// enums
Datatypes.RegisterDatatype(_eTcVn2dCodeSearchStrategy);
Datatypes.RegisterDatatype(_eTcVnAdaptiveThresholdMethod);
Datatypes.RegisterDatatype(_eTcVnBarcodeSearchDirection);
Datatypes.RegisterDatatype(_eTcVnBarcodeType);
Datatypes.RegisterDatatype(_eTcVnBlobCombination);
Datatypes.RegisterDatatype(_eTcVnBoostClassifierType);
Datatypes.RegisterDatatype(_eTcVnBorderInterpolationMethod);
Datatypes.RegisterDatatype(_eTcVnCalibrationPattern);
Datatypes.RegisterDatatype(_eTcVnCalibrationPatternOrigin);
Datatypes.RegisterDatatype(_eTcVnCameraState);
Datatypes.RegisterDatatype(_eTcVnClusteringAlgorithm);
Datatypes.RegisterDatatype(_eTcVnCodeDetectionModel);
Datatypes.RegisterDatatype(_eTcVnCodeType);
Datatypes.RegisterDatatype(_eTcVnColorMap);
Datatypes.RegisterDatatype(_eTcVnColorMapSize);
Datatypes.RegisterDatatype(_eTcVnColorSpaceTransform);
Datatypes.RegisterDatatype(_eTcVnColorTrainingMethod);
Datatypes.RegisterDatatype(_eTcVnConnectedComponentsAlgorithm);
Datatypes.RegisterDatatype(_eTcVnContainerExportFormat);
Datatypes.RegisterDatatype(_eTcVnContourApproximationMethod);
Datatypes.RegisterDatatype(_eTcVnContourRetrievalMode);
Datatypes.RegisterDatatype(_eTcVnContoursMatchComparisonMethod);
Datatypes.RegisterDatatype(_eTcVnDiffusivityTypeKAZE);
Datatypes.RegisterDatatype(_eTcVnDistanceTransformationLabel);
Datatypes.RegisterDatatype(_eTcVnDistanceTransformationMask);
Datatypes.RegisterDatatype(_eTcVnDistanceType);
Datatypes.RegisterDatatype(_eTcVnDrawMatchesFlags);
Datatypes.RegisterDatatype(_eTcVnDrawShape);
Datatypes.RegisterDatatype(_eTcVnEdgeDetectionAlgorithm);
Datatypes.RegisterDatatype(_eTcVnEdgeDirection);
Datatypes.RegisterDatatype(_eTcVnElementType);
Datatypes.RegisterDatatype(_eTcVnEstimationAlgorithm);
Datatypes.RegisterDatatype(_eTcVnExtremePointDirection);
Datatypes.RegisterDatatype(_eTcVnFeatureDescriptorTypeAKAZE);
Datatypes.RegisterDatatype(_eTcVnFeatureScalingType);
Datatypes.RegisterDatatype(_eTcVnFeatureScoreTypeORB);
Datatypes.RegisterDatatype(_eTcVnFilterDirection);
Datatypes.RegisterDatatype(_eTcVnFindTemplateWalshOptions);
Datatypes.RegisterDatatype(_eTcVnFlipAxis);
Datatypes.RegisterDatatype(_eTcVnFontType);
Datatypes.RegisterDatatype(_eTcVnHoughMethod);
Datatypes.RegisterDatatype(_eTcVnInitializableFunction);
Datatypes.RegisterDatatype(_eTcVnInterpolationType);
Datatypes.RegisterDatatype(_eTcVnKeypointDetectionTypeAGAST);
Datatypes.RegisterDatatype(_eTcVnKeypointDetectionTypeFAST);
Datatypes.RegisterDatatype(_eTcVnKnn);
Datatypes.RegisterDatatype(_eTcVnLineType);
Datatypes.RegisterDatatype(_eTcVnMatchTemplateWalshOptions);
Datatypes.RegisterDatatype(_eTcVnMorphologicalOperator);
Datatypes.RegisterDatatype(_eTcVnNbc);
Datatypes.RegisterDatatype(_eTcVnNormalizationType);
Datatypes.RegisterDatatype(_eTcVnOcrModelType);
Datatypes.RegisterDatatype(_eTcVnOcrOptions);
Datatypes.RegisterDatatype(_eTcVnOrientationMethod);
Datatypes.RegisterDatatype(_eTcVnPaddingMode);
Datatypes.RegisterDatatype(_eTcVnPixelConnectivity);
Datatypes.RegisterDatatype(_eTcVnPixelEncoding);
Datatypes.RegisterDatatype(_eTcVnPixelPackMode);
Datatypes.RegisterDatatype(_eTcVnPrototypeClusterer);
Datatypes.RegisterDatatype(_eTcVnRectangleIntersection);
Datatypes.RegisterDatatype(_eTcVnRotationAngle);
Datatypes.RegisterDatatype(_eTcVnRTrees);
Datatypes.RegisterDatatype(_eTcVnSignedNormalization);
Datatypes.RegisterDatatype(_eTcVnSolvePnPMethod);
Datatypes.RegisterDatatype(_eTcVnSta);
Datatypes.RegisterDatatype(_eTcVnStructuringElementShape);
Datatypes.RegisterDatatype(_eTcVnSvm);
Datatypes.RegisterDatatype(_eTcVnSvmKernelType);
Datatypes.RegisterDatatype(_eTcVnSvmSgdClassifierMarginType);
Datatypes.RegisterDatatype(_eTcVnSvmSgdClassifierType);
Datatypes.RegisterDatatype(_eTcVnTemplateMatchMethod);
Datatypes.RegisterDatatype(_eTcVnThresholdType);
Datatypes.RegisterDatatype(_eTcVnTimestamp);
Datatypes.RegisterDatatype(_eTcVnVectorCompareMethod);
Datatypes.RegisterDatatype(_eTcVnWorldCoordinateSystem);
Datatypes.RegisterDatatype(_eTcWatchdogAccumulationType);
Datatypes.RegisterDatatype(_gEV_CAMERA_STATE);
Datatypes.RegisterDatatype(_eTcVnDataLayout);
Datatypes.RegisterDatatype(_eTcVnReduceType);
Datatypes.RegisterDatatype(_eTcVnCircularityCalculationMethod);
Datatypes.RegisterDatatype(_eTcVnDataMatrixOptions);
Datatypes.RegisterDatatype(_eTcVnLayerNameType);
    
Datatypes.RegisterDatatype(_eTcVnComparisonOperator);
Datatypes.RegisterDatatype(_eTcVnDetectBarcodesWalshOptions);
Datatypes.RegisterDatatype(_eTcVnDetectPatternPointsOptions);
Datatypes.RegisterDatatype(_eTcVnDotCodeOptions);
Datatypes.RegisterDatatype(_eTcVnEdgeSelection);
Datatypes.RegisterDatatype(_eTcVnFindRoisMethod);
Datatypes.RegisterDatatype(_eTcVnJpegSampling);
Datatypes.RegisterDatatype(_eTcVnMergeRegionsOptions);
Datatypes.RegisterDatatype(_eTcVnPolarizedImageInterpolation);
Datatypes.RegisterDatatype(_eTcVnSalientFeaturesMethod);
// structs
Datatypes.RegisterDatatype(_gVSP_IMAGE_INFO);
Datatypes.RegisterDatatype(_gVSP_LEADER_PAYLOAD_IMAGE);
Datatypes.RegisterDatatype(_gVSP_PIXEL_FORMAT);
Datatypes.RegisterDatatype(_tcVnCameraCalibrationOptions);
Datatypes.RegisterDatatype(_tcVnCircularArc);
Datatypes.RegisterDatatype(_tcVnCodeGrades1D);
Datatypes.RegisterDatatype(_tcVnCodeGradesDM);
Datatypes.RegisterDatatype(_tcVnCodeGradesQR);
Datatypes.RegisterDatatype(_tcVnDMatch);
Datatypes.RegisterDatatype(_tcVnImageInfo);
Datatypes.RegisterDatatype(_tcVnKeyPoint);
//Datatypes.RegisterDatatype(_tcVnMatrix);
Datatypes.RegisterDatatype(_tcVnMoments);
Datatypes.RegisterDatatype(_tcVnParamsAGAST);
Datatypes.RegisterDatatype(_tcVnParamsAKAZE);
Datatypes.RegisterDatatype(_tcVnParamsBlobDetection);
Datatypes.RegisterDatatype(_tcVnParamsBRISK);
Datatypes.RegisterDatatype(_tcVnParamsFAST);
Datatypes.RegisterDatatype(_tcVnParamsGFTT);
Datatypes.RegisterDatatype(_tcVnParamsKAZE);
Datatypes.RegisterDatatype(_tcVnParamsMSER);
Datatypes.RegisterDatatype(_tcVnParamsORB);
Datatypes.RegisterDatatype(_tcVnParamsSB);
Datatypes.RegisterDatatype(_tcVnPixelFormat);
Datatypes.RegisterDatatype(_tcVnRectangle_DINT);
Datatypes.RegisterDatatype(_tcVnRectangle_UDINT);
Datatypes.RegisterDatatype(_tcVnRotatedRectangle);
Datatypes.RegisterDatatype(_tcVnSize2_REAL);

Datatypes.RegisterDatatype(_gVCP_ADDRESS_VALUE_PAIR);
Datatypes.RegisterDatatype(_tcVnSize2_DINT);
Datatypes.RegisterDatatype(_tcVnParamsFindRois);
Datatypes.RegisterDatatype(_tcVnParamsWalshBarcodeDetection);
// interfaces
Datatypes.RegisterDatatype(_iTcVnImage);
Datatypes.RegisterDatatype(_iTcVnContainer);
Datatypes.RegisterDatatype(_iTcVnDisplayableImage);
END_METHOD

END_FUNCTION_BLOCK

// ---- Datatypes/Aliases/_GVCP_REGISTER_VALUE.TcPOU
{attribute 'linkalways'}
{attribute 'no_explicit_call' := 'This FB is a CLASS and must be accessed using methods or properties'}
{attribute 'enable_dynamic_creation'}
FUNCTION_BLOCK _GVCP_REGISTER_VALUE EXTENDS AliasDatatypeBase
VAR
	localData : GVCP_REGISTER_VALUE;
	activeData : REFERENCE TO GVCP_REGISTER_VALUE REF= localData;
	aliasBaseDatatype : _UDINT(0);
END_VAR

PROPERTY PUBLIC Address : PVOID
GET
Address := ADR(activeData);
END_GET
END_PROPERTY

METHOD PUBLIC ClearReference
VAR_INPUT
END_VAR
activeData REF= localData;
SetBaseDatatypeReference();
END_METHOD

METHOD PUBLIC Clone : I_Datatype
VAR
    pClone : POINTER TO _GVCP_REGISTER_VALUE;
END_VAR
pClone := __NEW(_GVCP_REGISTER_VALUE(InitialValue := Value));
IF pClone = 0 THEN
    RETURN;
END_IF
pClone^.TryCopyFrom(THIS^);
Clone := pClone^;
END_METHOD

METHOD FB_init : BOOL
VAR_INPUT
	bInitRetains : BOOL; // if TRUE, the retain variables are initialized (warm start / cold start)
	bInCopyCode : BOOL;  // if TRUE, the instance afterwards gets moved into the copy code (online change)
	InitialValue : GVCP_REGISTER_VALUE := 0;
END_VAR
localData := InitialValue;
SetBaseDatatypeReference();
AddBaseDatatype(aliasBaseDatatype);
END_METHOD

PROPERTY PUBLIC Identifier : T_MAXSTRING
GET
Identifier := 'GVCP_REGISTER_VALUE';
END_GET
END_PROPERTY

METHOD PUBLIC MakeReferenceTo
VAR_INPUT
	ReferenceTarget : REFERENCE TO GVCP_REGISTER_VALUE;
END_VAR
activeData REF= ReferenceTarget;
SetBaseDatatypeReference();
END_METHOD

METHOD PROTECTED SetBaseDatatypeReference
VAR_INPUT
END_VAR
aliasBaseDatatype.MakeReferenceTo(activeData);
END_METHOD

PROPERTY PUBLIC Size : UDINT
GET
Size := SIZEOF(activeData);
END_GET
END_PROPERTY

METHOD TryMakeReferenceTo : BOOL
VAR_INPUT
	Target : I_Datatype;
END_VAR
VAR
	pTargetData : POINTER TO GVCP_REGISTER_VALUE;
END_VAR
IF NOT IsEquivalentTo(Target) THEN
	RETURN;
END_IF

pTargetData := Target.Address;
activeData REF= pTargetData^;
SetBaseDatatypeReference();
TryMakeReferenceTo := TRUE;
END_METHOD

PROPERTY PUBLIC Value : REFERENCE TO GVCP_REGISTER_VALUE
GET
Value REF= activeData;
END_GET
END_PROPERTY

END_FUNCTION_BLOCK

// ---- Datatypes/Enums/_ETcVnComparisonOperator.TcPOU
{attribute 'linkalways'}
{attribute 'no_explicit_call' := 'This FB is a CLASS and must be accessed using methods or properties'}
{attribute 'enable_dynamic_creation'}
FUNCTION_BLOCK _ETcVnComparisonOperator EXTENDS EnumDatatypeBase
VAR
	localData : ETcVnComparisonOperator;
	activeData : REFERENCE TO ETcVnComparisonOperator;
	enumBaseDatatype : _INT(localData);
END_VAR

METHOD PRIVATE AddLocalEnumeration
VAR_INPUT
	Enumeration : T_MAXSTRING;
	Value : ETcVnComparisonOperator;
END_VAR
AddEnumeration(Enumeration, Value);
END_METHOD

PROPERTY PUBLIC Address : PVOID
GET
Address := ADR(activeData);
END_GET
END_PROPERTY

METHOD PUBLIC ClearReference
VAR_INPUT
END_VAR
activeData REF= localData;
SetBaseDatatypeReference();
END_METHOD

METHOD PUBLIC Clone : I_Datatype
VAR
    pClone : POINTER TO _ETcVnComparisonOperator;
END_VAR
pClone := __NEW(_ETcVnComparisonOperator(InitialValue := Value));
IF pClone = 0 THEN
    RETURN;
END_IF
Clone := pClone^;
END_METHOD

METHOD FB_init : BOOL
VAR_INPUT
	bInitRetains : BOOL; // if TRUE, the retain variables are initialized (warm start / cold start)
	bInCopyCode : BOOL;  // if TRUE, the instance afterwards gets moved into the copy code (online change)
	InitialValue : ETcVnComparisonOperator;
END_VAR
localData := InitialValue;
AddBaseDatatype(enumBaseDatatype);
ClearReference();

AddLocalEnumeration('TCVN_CO_LESS', ETcVnComparisonOperator.TCVN_CO_LESS);
AddLocalEnumeration('TCVN_CO_GREATER', ETcVnComparisonOperator.TCVN_CO_GREATER);
END_METHOD

PROPERTY PUBLIC Identifier : T_MAXSTRING
GET
Identifier := 'ETcVnComparisonOperator';
END_GET
END_PROPERTY

METHOD IsEnumeratorValueEqual : BOOL
VAR_INPUT
	Enumerator : I_KeyValueForwardEnumerator;
END_VAR
VAR
	storedValue : ETcVnComparisonOperator;
END_VAR
IF NOT Enumerator.TryGet(storedValue) THEN
	RETURN;
END_IF

IsEnumeratorValueEqual := storedValue = activeData;
END_METHOD

METHOD PUBLIC MakeReferenceTo
VAR_INPUT
	ReferenceTarget : REFERENCE TO ETcVnComparisonOperator;
END_VAR
activeData REF= ReferenceTarget;
SetBaseDatatypeReference();
END_METHOD

METHOD PROTECTED SetBaseDatatypeReference
VAR_INPUT
END_VAR
enumBaseDatatype.MakeReferenceTo(activeData);
END_METHOD

PROPERTY PUBLIC Size : UDINT
GET
Size := SIZEOF(activeData);
END_GET
END_PROPERTY

METHOD TryMakeReferenceTo : BOOL
VAR_INPUT
	Target : I_Datatype;
END_VAR
VAR
	pTargetData : POINTER TO ETcVnComparisonOperator;
END_VAR
IF NOT IsEquivalentTo(Target) THEN
	RETURN;
END_IF

pTargetData := Target.Address;
activeData REF= pTargetData^;
SetBaseDatatypeReference();
TryMakeReferenceTo := TRUE;
END_METHOD

PROPERTY PUBLIC Value : ETcVnComparisonOperator
GET
Value := activeData;
END_GET
SET
activeData := Value;
END_SET
END_PROPERTY

END_FUNCTION_BLOCK

// ---- Datatypes/Enums/_ETcVnDetectBarcodesWalshOptions.TcPOU
{attribute 'linkalways'}
{attribute 'no_explicit_call' := 'This FB is a CLASS and must be accessed using methods or properties'}
{attribute 'enable_dynamic_creation'}
FUNCTION_BLOCK _ETcVnDetectBarcodesWalshOptions EXTENDS EnumDatatypeBase
VAR
	localData : ETcVnDetectBarcodesWalshOptions;
	activeData : REFERENCE TO ETcVnDetectBarcodesWalshOptions;
	enumBaseDatatype : _UDINT(localData);
END_VAR

METHOD PRIVATE AddLocalEnumeration
VAR_INPUT
	Enumeration : T_MAXSTRING;
	Value : ETcVnDetectBarcodesWalshOptions;
END_VAR
AddEnumeration(Enumeration, Value);
END_METHOD

PROPERTY PUBLIC Address : PVOID
GET
Address := ADR(activeData);
END_GET
END_PROPERTY

METHOD PUBLIC ClearReference
VAR_INPUT
END_VAR
activeData REF= localData;
SetBaseDatatypeReference();
END_METHOD

METHOD PUBLIC Clone : I_Datatype
VAR
    pClone : POINTER TO _ETcVnDetectBarcodesWalshOptions;
END_VAR
pClone := __NEW(_ETcVnDetectBarcodesWalshOptions(InitialValue := Value));
IF pClone = 0 THEN
    RETURN;
END_IF
Clone := pClone^;
END_METHOD

METHOD FB_init : BOOL
VAR_INPUT
	bInitRetains : BOOL; // if TRUE, the retain variables are initialized (warm start / cold start)
	bInCopyCode : BOOL;  // if TRUE, the instance afterwards gets moved into the copy code (online change)
	InitialValue : ETcVnDetectBarcodesWalshOptions;
END_VAR
localData := InitialValue;
AddBaseDatatype(enumBaseDatatype);
ClearReference();

AddLocalEnumeration('TCVN_DBWO_HORIZONTAL', ETcVnDetectBarcodesWalshOptions.TCVN_DBWO_HORIZONTAL);
AddLocalEnumeration('TCVN_DBWO_VERTICAL', ETcVnDetectBarcodesWalshOptions.TCVN_DBWO_VERTICAL);
AddLocalEnumeration('TCVN_DBWO_DIAGONAL_45', ETcVnDetectBarcodesWalshOptions.TCVN_DBWO_DIAGONAL_45);
AddLocalEnumeration('TCVN_DBWO_DIAGONAL_135', ETcVnDetectBarcodesWalshOptions.TCVN_DBWO_DIAGONAL_135);
AddLocalEnumeration('TCVN_DBWO_ALL_DIRECTIONS', ETcVnDetectBarcodesWalshOptions.TCVN_DBWO_ALL_DIRECTIONS);
END_METHOD

PROPERTY PUBLIC Identifier : T_MAXSTRING
GET
Identifier := 'ETcVnDetectBarcodesWalshOptions';
END_GET
END_PROPERTY

METHOD IsEnumeratorValueEqual : BOOL
VAR_INPUT
	Enumerator : I_KeyValueForwardEnumerator;
END_VAR
VAR
	storedValue : ETcVnDetectBarcodesWalshOptions;
END_VAR
IF NOT Enumerator.TryGet(storedValue) THEN
	RETURN;
END_IF

IsEnumeratorValueEqual := storedValue = activeData;
END_METHOD

METHOD PUBLIC MakeReferenceTo
VAR_INPUT
	ReferenceTarget : REFERENCE TO ETcVnDetectBarcodesWalshOptions;
END_VAR
activeData REF= ReferenceTarget;
SetBaseDatatypeReference();
END_METHOD

METHOD PROTECTED SetBaseDatatypeReference
VAR_INPUT
END_VAR
enumBaseDatatype.MakeReferenceTo(activeData);
END_METHOD

PROPERTY PUBLIC Size : UDINT
GET
Size := SIZEOF(activeData);
END_GET
END_PROPERTY

METHOD TryMakeReferenceTo : BOOL
VAR_INPUT
	Target : I_Datatype;
END_VAR
VAR
	pTargetData : POINTER TO ETcVnDetectBarcodesWalshOptions;
END_VAR
IF NOT IsEquivalentTo(Target) THEN
	RETURN;
END_IF

pTargetData := Target.Address;
activeData REF= pTargetData^;
SetBaseDatatypeReference();
TryMakeReferenceTo := TRUE;
END_METHOD

PROPERTY PUBLIC Value : ETcVnDetectBarcodesWalshOptions
GET
Value := activeData;
END_GET
SET
activeData := Value;
END_SET
END_PROPERTY

END_FUNCTION_BLOCK

// ---- Datatypes/Enums/_ETcVnDetectPatternPointsOptions.TcPOU
{attribute 'linkalways'}
{attribute 'no_explicit_call' := 'This FB is a CLASS and must be accessed using methods or properties'}
{attribute 'enable_dynamic_creation'}
FUNCTION_BLOCK _ETcVnDetectPatternPointsOptions EXTENDS EnumDatatypeBase
VAR
	localData : ETcVnDetectPatternPointsOptions;
	activeData : REFERENCE TO ETcVnDetectPatternPointsOptions;
	enumBaseDatatype : _UDINT(localData);
END_VAR

METHOD PRIVATE AddLocalEnumeration
VAR_INPUT
	Enumeration : T_MAXSTRING;
	Value : ETcVnDetectPatternPointsOptions;
END_VAR
AddEnumeration(Enumeration, Value);
END_METHOD

PROPERTY PUBLIC Address : PVOID
GET
Address := ADR(activeData);
END_GET
END_PROPERTY

METHOD PUBLIC ClearReference
VAR_INPUT
END_VAR
activeData REF= localData;
SetBaseDatatypeReference();
END_METHOD

METHOD PUBLIC Clone : I_Datatype
VAR
    pClone : POINTER TO _ETcVnDetectPatternPointsOptions;
END_VAR
pClone := __NEW(_ETcVnDetectPatternPointsOptions(InitialValue := Value));
IF pClone = 0 THEN
    RETURN;
END_IF
Clone := pClone^;
END_METHOD

METHOD FB_init : BOOL
VAR_INPUT
	bInitRetains : BOOL; // if TRUE, the retain variables are initialized (warm start / cold start)
	bInCopyCode : BOOL;  // if TRUE, the instance afterwards gets moved into the copy code (online change)
	InitialValue : ETcVnDetectPatternPointsOptions;
END_VAR
localData := InitialValue;
AddBaseDatatype(enumBaseDatatype);
ClearReference();

AddLocalEnumeration('TCVN_DPPO_SYMMETRIC', ETcVnDetectPatternPointsOptions.TCVN_DPPO_SYMMETRIC);
AddLocalEnumeration('TCVN_DPPO_ASYMMETRIC', ETcVnDetectPatternPointsOptions.TCVN_DPPO_ASYMMETRIC);
AddLocalEnumeration('TCVN_DPPO_CLUSTERING', ETcVnDetectPatternPointsOptions.TCVN_DPPO_CLUSTERING);
END_METHOD

PROPERTY PUBLIC Identifier : T_MAXSTRING
GET
Identifier := 'ETcVnDetectPatternPointsOptions';
END_GET
END_PROPERTY

METHOD IsEnumeratorValueEqual : BOOL
VAR_INPUT
	Enumerator : I_KeyValueForwardEnumerator;
END_VAR
VAR
	storedValue : ETcVnDetectPatternPointsOptions;
END_VAR
IF NOT Enumerator.TryGet(storedValue) THEN
	RETURN;
END_IF

IsEnumeratorValueEqual := storedValue = activeData;
END_METHOD

METHOD PUBLIC MakeReferenceTo
VAR_INPUT
	ReferenceTarget : REFERENCE TO ETcVnDetectPatternPointsOptions;
END_VAR
activeData REF= ReferenceTarget;
SetBaseDatatypeReference();
END_METHOD

METHOD PROTECTED SetBaseDatatypeReference
VAR_INPUT
END_VAR
enumBaseDatatype.MakeReferenceTo(activeData);
END_METHOD

PROPERTY PUBLIC Size : UDINT
GET
Size := SIZEOF(activeData);
END_GET
END_PROPERTY

METHOD TryMakeReferenceTo : BOOL
VAR_INPUT
	Target : I_Datatype;
END_VAR
VAR
	pTargetData : POINTER TO ETcVnDetectPatternPointsOptions;
END_VAR
IF NOT IsEquivalentTo(Target) THEN
	RETURN;
END_IF

pTargetData := Target.Address;
activeData REF= pTargetData^;
SetBaseDatatypeReference();
TryMakeReferenceTo := TRUE;
END_METHOD

PROPERTY PUBLIC Value : ETcVnDetectPatternPointsOptions
GET
Value := activeData;
END_GET
SET
activeData := Value;
END_SET
END_PROPERTY

END_FUNCTION_BLOCK

// ---- Datatypes/Enums/_ETcVnDotCodeOptions.TcPOU
{attribute 'linkalways'}
{attribute 'no_explicit_call' := 'This FB is a CLASS and must be accessed using methods or properties'}
{attribute 'enable_dynamic_creation'}
FUNCTION_BLOCK _ETcVnDotCodeOptions EXTENDS EnumDatatypeBase
VAR
	localData : ETcVnDotCodeOptions;
	activeData : REFERENCE TO ETcVnDotCodeOptions;
	enumBaseDatatype : _ULINT(localData);
END_VAR

METHOD PRIVATE AddLocalEnumeration
VAR_INPUT
	Enumeration : T_MAXSTRING;
	Value : ETcVnDotCodeOptions;
END_VAR
AddEnumeration(Enumeration, Value);
END_METHOD

PROPERTY PUBLIC Address : PVOID
GET
Address := ADR(activeData);
END_GET
END_PROPERTY

METHOD PUBLIC ClearReference
VAR_INPUT
END_VAR
activeData REF= localData;
SetBaseDatatypeReference();
END_METHOD

METHOD PUBLIC Clone : I_Datatype
VAR
    pClone : POINTER TO _ETcVnDotCodeOptions;
END_VAR
pClone := __NEW(_ETcVnDotCodeOptions(InitialValue := Value));
IF pClone = 0 THEN
    RETURN;
END_IF
Clone := pClone^;
END_METHOD

METHOD FB_init : BOOL
VAR_INPUT
	bInitRetains : BOOL; // if TRUE, the retain variables are initialized (warm start / cold start)
	bInCopyCode : BOOL;  // if TRUE, the instance afterwards gets moved into the copy code (online change)
	InitialValue : ETcVnDotCodeOptions;
END_VAR
localData := InitialValue;
AddBaseDatatype(enumBaseDatatype);
ClearReference();

AddLocalEnumeration('TCVN_DCO_DEFAULT', ETcVnDotCodeOptions.TCVN_DCO_DEFAULT);
AddLocalEnumeration('TCVN_DCO_BINARY_INPUT', ETcVnDotCodeOptions.TCVN_DCO_BINARY_INPUT);
AddLocalEnumeration('TCVN_DCO_DETECTBLOBS', ETcVnDotCodeOptions.TCVN_DCO_DETECTBLOBS);
AddLocalEnumeration('TCVN_DCO_FILTERCONTOURS', ETcVnDotCodeOptions.TCVN_DCO_FILTERCONTOURS);
AddLocalEnumeration('TCVN_DCO_REGULAR_COLOR', ETcVnDotCodeOptions.TCVN_DCO_REGULAR_COLOR);
AddLocalEnumeration('TCVN_DCO_INVERTED_COLOR', ETcVnDotCodeOptions.TCVN_DCO_INVERTED_COLOR);
END_METHOD

PROPERTY PUBLIC Identifier : T_MAXSTRING
GET
Identifier := 'ETcVnDotCodeOptions';
END_GET
END_PROPERTY

METHOD IsEnumeratorValueEqual : BOOL
VAR_INPUT
	Enumerator : I_KeyValueForwardEnumerator;
END_VAR
VAR
	storedValue : ETcVnDotCodeOptions;
END_VAR
IF NOT Enumerator.TryGet(storedValue) THEN
	RETURN;
END_IF

IsEnumeratorValueEqual := storedValue = activeData;
END_METHOD

METHOD PUBLIC MakeReferenceTo
VAR_INPUT
	ReferenceTarget : REFERENCE TO ETcVnDotCodeOptions;
END_VAR
activeData REF= ReferenceTarget;
SetBaseDatatypeReference();
END_METHOD

METHOD PROTECTED SetBaseDatatypeReference
VAR_INPUT
END_VAR
enumBaseDatatype.MakeReferenceTo(activeData);
END_METHOD

PROPERTY PUBLIC Size : UDINT
GET
Size := SIZEOF(activeData);
END_GET
END_PROPERTY

METHOD TryMakeReferenceTo : BOOL
VAR_INPUT
	Target : I_Datatype;
END_VAR
VAR
	pTargetData : POINTER TO ETcVnDotCodeOptions;
END_VAR
IF NOT IsEquivalentTo(Target) THEN
	RETURN;
END_IF

pTargetData := Target.Address;
activeData REF= pTargetData^;
SetBaseDatatypeReference();
TryMakeReferenceTo := TRUE;
END_METHOD

PROPERTY PUBLIC Value : ETcVnDotCodeOptions
GET
Value := activeData;
END_GET
SET
activeData := Value;
END_SET
END_PROPERTY

END_FUNCTION_BLOCK

// ---- Datatypes/Enums/_ETcVnEdgeSelection.TcPOU
{attribute 'linkalways'}
{attribute 'no_explicit_call' := 'This FB is a CLASS and must be accessed using methods or properties'}
{attribute 'enable_dynamic_creation'}
FUNCTION_BLOCK _ETcVnEdgeSelection EXTENDS EnumDatatypeBase
VAR
	localData : ETcVnEdgeSelection;
	activeData : REFERENCE TO ETcVnEdgeSelection;
	enumBaseDatatype : _DINT(localData);
END_VAR

METHOD PRIVATE AddLocalEnumeration
VAR_INPUT
	Enumeration : T_MAXSTRING;
	Value : ETcVnEdgeSelection;
END_VAR
AddEnumeration(Enumeration, Value);
END_METHOD

PROPERTY PUBLIC Address : PVOID
GET
Address := ADR(activeData);
END_GET
END_PROPERTY

METHOD PUBLIC ClearReference
VAR_INPUT
END_VAR
activeData REF= localData;
SetBaseDatatypeReference();
END_METHOD

METHOD PUBLIC Clone : I_Datatype
VAR
    pClone : POINTER TO _ETcVnEdgeSelection;
END_VAR
pClone := __NEW(_ETcVnEdgeSelection(InitialValue := Value));
IF pClone = 0 THEN
    RETURN;
END_IF
Clone := pClone^;
END_METHOD

METHOD FB_init : BOOL
VAR_INPUT
	bInitRetains : BOOL; // if TRUE, the retain variables are initialized (warm start / cold start)
	bInCopyCode : BOOL;  // if TRUE, the instance afterwards gets moved into the copy code (online change)
	InitialValue : ETcVnEdgeSelection;
END_VAR
localData := InitialValue;
AddBaseDatatype(enumBaseDatatype);
ClearReference();

AddLocalEnumeration('TCVN_ES_RISING', ETcVnEdgeSelection.TCVN_ES_RISING);
AddLocalEnumeration('TCVN_ES_FALLING', ETcVnEdgeSelection.TCVN_ES_FALLING);
AddLocalEnumeration('TCVN_ES_ANY', ETcVnEdgeSelection.TCVN_ES_ANY);
END_METHOD

PROPERTY PUBLIC Identifier : T_MAXSTRING
GET
Identifier := 'ETcVnEdgeSelection';
END_GET
END_PROPERTY

METHOD IsEnumeratorValueEqual : BOOL
VAR_INPUT
	Enumerator : I_KeyValueForwardEnumerator;
END_VAR
VAR
	storedValue : ETcVnEdgeSelection;
END_VAR
IF NOT Enumerator.TryGet(storedValue) THEN
	RETURN;
END_IF

IsEnumeratorValueEqual := storedValue = activeData;
END_METHOD

METHOD PUBLIC MakeReferenceTo
VAR_INPUT
	ReferenceTarget : REFERENCE TO ETcVnEdgeSelection;
END_VAR
activeData REF= ReferenceTarget;
SetBaseDatatypeReference();
END_METHOD

METHOD PROTECTED SetBaseDatatypeReference
VAR_INPUT
END_VAR
enumBaseDatatype.MakeReferenceTo(activeData);
END_METHOD

PROPERTY PUBLIC Size : UDINT
GET
Size := SIZEOF(activeData);
END_GET
END_PROPERTY

METHOD TryMakeReferenceTo : BOOL
VAR_INPUT
	Target : I_Datatype;
END_VAR
VAR
	pTargetData : POINTER TO ETcVnEdgeSelection;
END_VAR
IF NOT IsEquivalentTo(Target) THEN
	RETURN;
END_IF

pTargetData := Target.Address;
activeData REF= pTargetData^;
SetBaseDatatypeReference();
TryMakeReferenceTo := TRUE;
END_METHOD

PROPERTY PUBLIC Value : ETcVnEdgeSelection
GET
Value := activeData;
END_GET
SET
activeData := Value;
END_SET
END_PROPERTY

END_FUNCTION_BLOCK

// ---- Datatypes/Enums/_ETcVnFindRoisMethod.TcPOU
{attribute 'linkalways'}
{attribute 'no_explicit_call' := 'This FB is a CLASS and must be accessed using methods or properties'}
{attribute 'enable_dynamic_creation'}
FUNCTION_BLOCK _ETcVnFindRoisMethod EXTENDS EnumDatatypeBase
VAR
	localData : ETcVnFindRoisMethod;
	activeData : REFERENCE TO ETcVnFindRoisMethod;
	enumBaseDatatype : _UDINT(localData);
END_VAR

METHOD PRIVATE AddLocalEnumeration
VAR_INPUT
	Enumeration : T_MAXSTRING;
	Value : ETcVnFindRoisMethod;
END_VAR
AddEnumeration(Enumeration, Value);
END_METHOD

PROPERTY PUBLIC Address : PVOID
GET
Address := ADR(activeData);
END_GET
END_PROPERTY

METHOD PUBLIC ClearReference
VAR_INPUT
END_VAR
activeData REF= localData;
SetBaseDatatypeReference();
END_METHOD

METHOD PUBLIC Clone : I_Datatype
VAR
    pClone : POINTER TO _ETcVnFindRoisMethod;
END_VAR
pClone := __NEW(_ETcVnFindRoisMethod(InitialValue := Value));
IF pClone = 0 THEN
    RETURN;
END_IF
Clone := pClone^;
END_METHOD

METHOD FB_init : BOOL
VAR_INPUT
	bInitRetains : BOOL; // if TRUE, the retain variables are initialized (warm start / cold start)
	bInCopyCode : BOOL;  // if TRUE, the instance afterwards gets moved into the copy code (online change)
	InitialValue : ETcVnFindRoisMethod;
END_VAR
localData := InitialValue;
AddBaseDatatype(enumBaseDatatype);
ClearReference();

AddLocalEnumeration('TCVN_FRM_GRID', ETcVnFindRoisMethod.TCVN_FRM_GRID);
AddLocalEnumeration('TCVN_FRM_CONNECTEDCOMPONENTS', ETcVnFindRoisMethod.TCVN_FRM_CONNECTEDCOMPONENTS);
END_METHOD

PROPERTY PUBLIC Identifier : T_MAXSTRING
GET
Identifier := 'ETcVnFindRoisMethod';
END_GET
END_PROPERTY

METHOD IsEnumeratorValueEqual : BOOL
VAR_INPUT
	Enumerator : I_KeyValueForwardEnumerator;
END_VAR
VAR
	storedValue : ETcVnFindRoisMethod;
END_VAR
IF NOT Enumerator.TryGet(storedValue) THEN
	RETURN;
END_IF

IsEnumeratorValueEqual := storedValue = activeData;
END_METHOD

METHOD PUBLIC MakeReferenceTo
VAR_INPUT
	ReferenceTarget : REFERENCE TO ETcVnFindRoisMethod;
END_VAR
activeData REF= ReferenceTarget;
SetBaseDatatypeReference();
END_METHOD

METHOD PROTECTED SetBaseDatatypeReference
VAR_INPUT
END_VAR
enumBaseDatatype.MakeReferenceTo(activeData);
END_METHOD

PROPERTY PUBLIC Size : UDINT
GET
Size := SIZEOF(activeData);
END_GET
END_PROPERTY

METHOD TryMakeReferenceTo : BOOL
VAR_INPUT
	Target : I_Datatype;
END_VAR
VAR
	pTargetData : POINTER TO ETcVnFindRoisMethod;
END_VAR
IF NOT IsEquivalentTo(Target) THEN
	RETURN;
END_IF

pTargetData := Target.Address;
activeData REF= pTargetData^;
SetBaseDatatypeReference();
TryMakeReferenceTo := TRUE;
END_METHOD

PROPERTY PUBLIC Value : ETcVnFindRoisMethod
GET
Value := activeData;
END_GET
SET
activeData := Value;
END_SET
END_PROPERTY

END_FUNCTION_BLOCK

// ---- Datatypes/Enums/_ETcVnJpegSampling.TcPOU
{attribute 'linkalways'}
{attribute 'no_explicit_call' := 'This FB is a CLASS and must be accessed using methods or properties'}
{attribute 'enable_dynamic_creation'}
FUNCTION_BLOCK _ETcVnJpegSampling EXTENDS EnumDatatypeBase
VAR
	localData : ETcVnJpegSampling;
	activeData : REFERENCE TO ETcVnJpegSampling;
	enumBaseDatatype : _DINT(localData);
END_VAR

METHOD PRIVATE AddLocalEnumeration
VAR_INPUT
	Enumeration : T_MAXSTRING;
	Value : ETcVnJpegSampling;
END_VAR
AddEnumeration(Enumeration, Value);
END_METHOD

PROPERTY PUBLIC Address : PVOID
GET
Address := ADR(activeData);
END_GET
END_PROPERTY

METHOD PUBLIC ClearReference
VAR_INPUT
END_VAR
activeData REF= localData;
SetBaseDatatypeReference();
END_METHOD

METHOD PUBLIC Clone : I_Datatype
VAR
    pClone : POINTER TO _ETcVnJpegSampling;
END_VAR
pClone := __NEW(_ETcVnJpegSampling(InitialValue := Value));
IF pClone = 0 THEN
    RETURN;
END_IF
Clone := pClone^;
END_METHOD

METHOD FB_init : BOOL
VAR_INPUT
	bInitRetains : BOOL; // if TRUE, the retain variables are initialized (warm start / cold start)
	bInCopyCode : BOOL;  // if TRUE, the instance afterwards gets moved into the copy code (online change)
	InitialValue : ETcVnJpegSampling;
END_VAR
localData := InitialValue;
AddBaseDatatype(enumBaseDatatype);
ClearReference();

AddLocalEnumeration('TCVN_JS_444', ETcVnJpegSampling.TCVN_JS_444);
AddLocalEnumeration('TCVN_JS_440', ETcVnJpegSampling.TCVN_JS_440);
AddLocalEnumeration('TCVN_JS_422', ETcVnJpegSampling.TCVN_JS_422);
AddLocalEnumeration('TCVN_JS_420', ETcVnJpegSampling.TCVN_JS_420);
AddLocalEnumeration('TCVN_JS_411', ETcVnJpegSampling.TCVN_JS_411);
AddLocalEnumeration('TCVN_JS_410', ETcVnJpegSampling.TCVN_JS_410);
END_METHOD

PROPERTY PUBLIC Identifier : T_MAXSTRING
GET
Identifier := 'ETcVnJpegSampling';
END_GET
END_PROPERTY

METHOD IsEnumeratorValueEqual : BOOL
VAR_INPUT
	Enumerator : I_KeyValueForwardEnumerator;
END_VAR
VAR
	storedValue : ETcVnJpegSampling;
END_VAR
IF NOT Enumerator.TryGet(storedValue) THEN
	RETURN;
END_IF

IsEnumeratorValueEqual := storedValue = activeData;
END_METHOD

METHOD PUBLIC MakeReferenceTo
VAR_INPUT
	ReferenceTarget : REFERENCE TO ETcVnJpegSampling;
END_VAR
activeData REF= ReferenceTarget;
SetBaseDatatypeReference();
END_METHOD

METHOD PROTECTED SetBaseDatatypeReference
VAR_INPUT
END_VAR
enumBaseDatatype.MakeReferenceTo(activeData);
END_METHOD

PROPERTY PUBLIC Size : UDINT
GET
Size := SIZEOF(activeData);
END_GET
END_PROPERTY

METHOD TryMakeReferenceTo : BOOL
VAR_INPUT
	Target : I_Datatype;
END_VAR
VAR
	pTargetData : POINTER TO ETcVnJpegSampling;
END_VAR
IF NOT IsEquivalentTo(Target) THEN
	RETURN;
END_IF

pTargetData := Target.Address;
activeData REF= pTargetData^;
SetBaseDatatypeReference();
TryMakeReferenceTo := TRUE;
END_METHOD

PROPERTY PUBLIC Value : ETcVnJpegSampling
GET
Value := activeData;
END_GET
SET
activeData := Value;
END_SET
END_PROPERTY

END_FUNCTION_BLOCK

// ---- Datatypes/Enums/_ETcVnMergeRegionsOptions.TcPOU
{attribute 'linkalways'}
{attribute 'no_explicit_call' := 'This FB is a CLASS and must be accessed using methods or properties'}
{attribute 'enable_dynamic_creation'}
FUNCTION_BLOCK _ETcVnMergeRegionsOptions EXTENDS EnumDatatypeBase
VAR
	localData : ETcVnMergeRegionsOptions;
	activeData : REFERENCE TO ETcVnMergeRegionsOptions;
	enumBaseDatatype : _ULINT(localData);
END_VAR

METHOD PRIVATE AddLocalEnumeration
VAR_INPUT
	Enumeration : T_MAXSTRING;
	Value : ETcVnMergeRegionsOptions;
END_VAR
AddEnumeration(Enumeration, Value);
END_METHOD

PROPERTY PUBLIC Address : PVOID
GET
Address := ADR(activeData);
END_GET
END_PROPERTY

METHOD PUBLIC ClearReference
VAR_INPUT
END_VAR
activeData REF= localData;
SetBaseDatatypeReference();
END_METHOD

METHOD PUBLIC Clone : I_Datatype
VAR
    pClone : POINTER TO _ETcVnMergeRegionsOptions;
END_VAR
pClone := __NEW(_ETcVnMergeRegionsOptions(InitialValue := Value));
IF pClone = 0 THEN
    RETURN;
END_IF
Clone := pClone^;
END_METHOD

METHOD FB_init : BOOL
VAR_INPUT
	bInitRetains : BOOL; // if TRUE, the retain variables are initialized (warm start / cold start)
	bInCopyCode : BOOL;  // if TRUE, the instance afterwards gets moved into the copy code (online change)
	InitialValue : ETcVnMergeRegionsOptions;
END_VAR
localData := InitialValue;
AddBaseDatatype(enumBaseDatatype);
ClearReference();

AddLocalEnumeration('TCVN_MRO_UPRIGHT_BOUNDING_RECT', ETcVnMergeRegionsOptions.TCVN_MRO_UPRIGHT_BOUNDING_RECT);
END_METHOD

PROPERTY PUBLIC Identifier : T_MAXSTRING
GET
Identifier := 'ETcVnMergeRegionsOptions';
END_GET
END_PROPERTY

METHOD IsEnumeratorValueEqual : BOOL
VAR_INPUT
	Enumerator : I_KeyValueForwardEnumerator;
END_VAR
VAR
	storedValue : ETcVnMergeRegionsOptions;
END_VAR
IF NOT Enumerator.TryGet(storedValue) THEN
	RETURN;
END_IF

IsEnumeratorValueEqual := storedValue = activeData;
END_METHOD

METHOD PUBLIC MakeReferenceTo
VAR_INPUT
	ReferenceTarget : REFERENCE TO ETcVnMergeRegionsOptions;
END_VAR
activeData REF= ReferenceTarget;
SetBaseDatatypeReference();
END_METHOD

METHOD PROTECTED SetBaseDatatypeReference
VAR_INPUT
END_VAR
enumBaseDatatype.MakeReferenceTo(activeData);
END_METHOD

PROPERTY PUBLIC Size : UDINT
GET
Size := SIZEOF(activeData);
END_GET
END_PROPERTY

METHOD TryMakeReferenceTo : BOOL
VAR_INPUT
	Target : I_Datatype;
END_VAR
VAR
	pTargetData : POINTER TO ETcVnMergeRegionsOptions;
END_VAR
IF NOT IsEquivalentTo(Target) THEN
	RETURN;
END_IF

pTargetData := Target.Address;
activeData REF= pTargetData^;
SetBaseDatatypeReference();
TryMakeReferenceTo := TRUE;
END_METHOD

PROPERTY PUBLIC Value : ETcVnMergeRegionsOptions
GET
Value := activeData;
END_GET
SET
activeData := Value;
END_SET
END_PROPERTY

END_FUNCTION_BLOCK

// ---- Datatypes/Enums/_ETcVnPolarizedImageInterpolation.TcPOU
{attribute 'linkalways'}
{attribute 'no_explicit_call' := 'This FB is a CLASS and must be accessed using methods or properties'}
{attribute 'enable_dynamic_creation'}
FUNCTION_BLOCK _ETcVnPolarizedImageInterpolation EXTENDS EnumDatatypeBase
VAR
	localData : ETcVnPolarizedImageInterpolation;
	activeData : REFERENCE TO ETcVnPolarizedImageInterpolation;
	enumBaseDatatype : _DINT(localData);
END_VAR

METHOD PRIVATE AddLocalEnumeration
VAR_INPUT
	Enumeration : T_MAXSTRING;
	Value : ETcVnPolarizedImageInterpolation;
END_VAR
AddEnumeration(Enumeration, Value);
END_METHOD

PROPERTY PUBLIC Address : PVOID
GET
Address := ADR(activeData);
END_GET
END_PROPERTY

METHOD PUBLIC ClearReference
VAR_INPUT
END_VAR
activeData REF= localData;
SetBaseDatatypeReference();
END_METHOD

METHOD PUBLIC Clone : I_Datatype
VAR
    pClone : POINTER TO _ETcVnPolarizedImageInterpolation;
END_VAR
pClone := __NEW(_ETcVnPolarizedImageInterpolation(InitialValue := Value));
IF pClone = 0 THEN
    RETURN;
END_IF
Clone := pClone^;
END_METHOD

METHOD FB_init : BOOL
VAR_INPUT
	bInitRetains : BOOL; // if TRUE, the retain variables are initialized (warm start / cold start)
	bInCopyCode : BOOL;  // if TRUE, the instance afterwards gets moved into the copy code (online change)
	InitialValue : ETcVnPolarizedImageInterpolation;
END_VAR
localData := InitialValue;
AddBaseDatatype(enumBaseDatatype);
ClearReference();

AddLocalEnumeration('TCVN_PII_NONE', ETcVnPolarizedImageInterpolation.TCVN_PII_NONE);
AddLocalEnumeration('TCVN_PII_NEAREST_NEIGHBOR', ETcVnPolarizedImageInterpolation.TCVN_PII_NEAREST_NEIGHBOR);
AddLocalEnumeration('TCVN_PII_BILINEAR', ETcVnPolarizedImageInterpolation.TCVN_PII_BILINEAR);
AddLocalEnumeration('TCVN_PII_BICUBIC', ETcVnPolarizedImageInterpolation.TCVN_PII_BICUBIC);
AddLocalEnumeration('TCVN_PII_LANCZOS4', ETcVnPolarizedImageInterpolation.TCVN_PII_LANCZOS4);
END_METHOD

PROPERTY PUBLIC Identifier : T_MAXSTRING
GET
Identifier := 'ETcVnPolarizedImageInterpolation';
END_GET
END_PROPERTY

METHOD IsEnumeratorValueEqual : BOOL
VAR_INPUT
	Enumerator : I_KeyValueForwardEnumerator;
END_VAR
VAR
	storedValue : ETcVnPolarizedImageInterpolation;
END_VAR
IF NOT Enumerator.TryGet(storedValue) THEN
	RETURN;
END_IF

IsEnumeratorValueEqual := storedValue = activeData;
END_METHOD

METHOD PUBLIC MakeReferenceTo
VAR_INPUT
	ReferenceTarget : REFERENCE TO ETcVnPolarizedImageInterpolation;
END_VAR
activeData REF= ReferenceTarget;
SetBaseDatatypeReference();
END_METHOD

METHOD PROTECTED SetBaseDatatypeReference
VAR_INPUT
END_VAR
enumBaseDatatype.MakeReferenceTo(activeData);
END_METHOD

PROPERTY PUBLIC Size : UDINT
GET
Size := SIZEOF(activeData);
END_GET
END_PROPERTY

METHOD TryMakeReferenceTo : BOOL
VAR_INPUT
	Target : I_Datatype;
END_VAR
VAR
	pTargetData : POINTER TO ETcVnPolarizedImageInterpolation;
END_VAR
IF NOT IsEquivalentTo(Target) THEN
	RETURN;
END_IF

pTargetData := Target.Address;
activeData REF= pTargetData^;
SetBaseDatatypeReference();
TryMakeReferenceTo := TRUE;
END_METHOD

PROPERTY PUBLIC Value : ETcVnPolarizedImageInterpolation
GET
Value := activeData;
END_GET
SET
activeData := Value;
END_SET
END_PROPERTY

END_FUNCTION_BLOCK

// ---- Datatypes/Enums/_ETcVnSalientFeaturesMethod.TcPOU
{attribute 'linkalways'}
{attribute 'no_explicit_call' := 'This FB is a CLASS and must be accessed using methods or properties'}
{attribute 'enable_dynamic_creation'}
FUNCTION_BLOCK _ETcVnSalientFeaturesMethod EXTENDS EnumDatatypeBase
VAR
	localData : ETcVnSalientFeaturesMethod;
	activeData : REFERENCE TO ETcVnSalientFeaturesMethod;
	enumBaseDatatype : _UDINT(localData);
END_VAR

METHOD PRIVATE AddLocalEnumeration
VAR_INPUT
	Enumeration : T_MAXSTRING;
	Value : ETcVnSalientFeaturesMethod;
END_VAR
AddEnumeration(Enumeration, Value);
END_METHOD

PROPERTY PUBLIC Address : PVOID
GET
Address := ADR(activeData);
END_GET
END_PROPERTY

METHOD PUBLIC ClearReference
VAR_INPUT
END_VAR
activeData REF= localData;
SetBaseDatatypeReference();
END_METHOD

METHOD PUBLIC Clone : I_Datatype
VAR
    pClone : POINTER TO _ETcVnSalientFeaturesMethod;
END_VAR
pClone := __NEW(_ETcVnSalientFeaturesMethod(InitialValue := Value));
IF pClone = 0 THEN
    RETURN;
END_IF
Clone := pClone^;
END_METHOD

METHOD FB_init : BOOL
VAR_INPUT
	bInitRetains : BOOL; // if TRUE, the retain variables are initialized (warm start / cold start)
	bInCopyCode : BOOL;  // if TRUE, the instance afterwards gets moved into the copy code (online change)
	InitialValue : ETcVnSalientFeaturesMethod;
END_VAR
localData := InitialValue;
AddBaseDatatype(enumBaseDatatype);
ClearReference();

AddLocalEnumeration('TCVN_SFM_WALSH_CODE', ETcVnSalientFeaturesMethod.TCVN_SFM_WALSH_CODE);
AddLocalEnumeration('TCVN_SFM_SOBEL', ETcVnSalientFeaturesMethod.TCVN_SFM_SOBEL);
END_METHOD

PROPERTY PUBLIC Identifier : T_MAXSTRING
GET
Identifier := 'ETcVnSalientFeaturesMethod';
END_GET
END_PROPERTY

METHOD IsEnumeratorValueEqual : BOOL
VAR_INPUT
	Enumerator : I_KeyValueForwardEnumerator;
END_VAR
VAR
	storedValue : ETcVnSalientFeaturesMethod;
END_VAR
IF NOT Enumerator.TryGet(storedValue) THEN
	RETURN;
END_IF

IsEnumeratorValueEqual := storedValue = activeData;
END_METHOD

METHOD PUBLIC MakeReferenceTo
VAR_INPUT
	ReferenceTarget : REFERENCE TO ETcVnSalientFeaturesMethod;
END_VAR
activeData REF= ReferenceTarget;
SetBaseDatatypeReference();
END_METHOD

METHOD PROTECTED SetBaseDatatypeReference
VAR_INPUT
END_VAR
enumBaseDatatype.MakeReferenceTo(activeData);
END_METHOD

PROPERTY PUBLIC Size : UDINT
GET
Size := SIZEOF(activeData);
END_GET
END_PROPERTY

METHOD TryMakeReferenceTo : BOOL
VAR_INPUT
	Target : I_Datatype;
END_VAR
VAR
	pTargetData : POINTER TO ETcVnSalientFeaturesMethod;
END_VAR
IF NOT IsEquivalentTo(Target) THEN
	RETURN;
END_IF

pTargetData := Target.Address;
activeData REF= pTargetData^;
SetBaseDatatypeReference();
TryMakeReferenceTo := TRUE;
END_METHOD

PROPERTY PUBLIC Value : ETcVnSalientFeaturesMethod
GET
Value := activeData;
END_GET
SET
activeData := Value;
END_SET
END_PROPERTY

END_FUNCTION_BLOCK

// ---- Datatypes/Structs/_GVCP_ADDRESS_VALUE_PAIR.TcPOU
{attribute 'linkalways'}
{attribute 'no_explicit_call' := 'This FB is a CLASS and must be accessed using methods or properties'}
{attribute 'enable_dynamic_creation'}
FUNCTION_BLOCK _GVCP_ADDRESS_VALUE_PAIR EXTENDS StructuredDatatypeBase
VAR
    localData : GVCP_ADDRESS_VALUE_PAIR;
    activeData : REFERENCE TO GVCP_ADDRESS_VALUE_PAIR REF= localData;
    _nAddress : _GVCP_REGISTER_ADDRESS(0);
    _nValue : _GVCP_REGISTER_VALUE(0);
END_VAR

PROPERTY PUBLIC Address : PVOID
GET
Address := ADR(activeData);
END_GET
END_PROPERTY

METHOD PUBLIC ClearReference
VAR_INPUT
END_VAR
activeData REF= localData;
SetMemberReference();
END_METHOD

METHOD PUBLIC Clone : I_Datatype
VAR
    pClone : POINTER TO _GVCP_ADDRESS_VALUE_PAIR;
END_VAR
pClone := __NEW(_GVCP_ADDRESS_VALUE_PAIR);
IF pClone = 0 THEN
    RETURN;
END_IF
pClone^.TryCopyFrom(THIS^);
Clone := pClone^;
END_METHOD

METHOD FB_init : BOOL
VAR_INPUT
	bInitRetains : BOOL; // if TRUE, the retain variables are initialized (warm start / cold start)
	bInCopyCode : BOOL;  // if TRUE, the instance afterwards gets moved into the copy code (online change)
END_VAR
SetMemberReference();
AddMember('nAddress', _nAddress);
AddMember('nValue', _nValue);
END_METHOD

PROPERTY PUBLIC Identifier : T_MAXSTRING
GET
Identifier := 'GVCP_ADDRESS_VALUE_PAIR';
END_GET
END_PROPERTY

METHOD PUBLIC MakeReferenceTo
VAR_INPUT
	ReferenceTarget : REFERENCE TO GVCP_ADDRESS_VALUE_PAIR;
END_VAR
activeData REF= ReferenceTarget;
SetMemberReference();
END_METHOD

PROPERTY PUBLIC nAddress : REFERENCE TO _GVCP_REGISTER_ADDRESS
GET
nAddress REF= _nAddress;
END_GET
END_PROPERTY

PROPERTY PUBLIC nValue : REFERENCE TO _GVCP_REGISTER_VALUE
GET
nValue REF= _nValue;
END_GET
END_PROPERTY

METHOD PROTECTED SetMemberReference
VAR_INPUT
END_VAR
_nAddress.MakeReferenceTo(activeData.nAddress);
_nValue.MakeReferenceTo(activeData.nValue);
END_METHOD

PROPERTY PUBLIC Size : UDINT
GET
Size := SIZEOF(activeData);
END_GET
END_PROPERTY

METHOD TryMakeReferenceTo : BOOL
VAR_INPUT
	Target : I_Datatype;
END_VAR
VAR
	pTargetData : POINTER TO GVCP_ADDRESS_VALUE_PAIR;
END_VAR
IF NOT IsEquivalentTo(Target) THEN
	RETURN;
END_IF

pTargetData := Target.Address;
activeData REF= pTargetData^;
SetMemberReference();
TryMakeReferenceTo := TRUE;
END_METHOD

PROPERTY PUBLIC Value : REFERENCE TO GVCP_ADDRESS_VALUE_PAIR
GET
Value REF= activeData;
END_GET
END_PROPERTY

END_FUNCTION_BLOCK

// ---- Datatypes/Structs/_TcVnSize2_DINT.TcPOU
{attribute 'linkalways'}
{attribute 'no_explicit_call' := 'This FB is a CLASS and must be accessed using methods or properties'}
{attribute 'enable_dynamic_creation'}
FUNCTION_BLOCK _TcVnSize2_DINT EXTENDS StructuredDatatypeBase
VAR
    localData : TcVnSize2_DINT;
    activeData : REFERENCE TO TcVnSize2_DINT REF= localData;
    _nWidth : _DINT(localData.nWidth);
    _nHeight : _DINT(localData.nHeight);
END_VAR

PROPERTY PUBLIC Address : PVOID
GET
Address := ADR(activeData);
END_GET
END_PROPERTY

METHOD PUBLIC ClearReference
VAR_INPUT
END_VAR
activeData REF= localData;
SetMemberReference();
END_METHOD

METHOD PUBLIC Clone : I_Datatype
VAR
    pClone : POINTER TO _TcVnSize2_DINT;
END_VAR
pClone := __NEW(_TcVnSize2_DINT);
IF pClone = 0 THEN
    RETURN;
END_IF
pClone^.TryCopyFrom(THIS^);
Clone := pClone^;
END_METHOD

METHOD FB_init : BOOL
VAR_INPUT
	bInitRetains : BOOL; // if TRUE, the retain variables are initialized (warm start / cold start)
	bInCopyCode : BOOL;  // if TRUE, the instance afterwards gets moved into the copy code (online change)
END_VAR
SetMemberReference();
AddMember('nWidth', _nWidth);
AddMember('nHeight', _nHeight);
END_METHOD

PROPERTY PUBLIC Identifier : T_MAXSTRING
GET
Identifier := 'TcVnSize2_DINT';
END_GET
END_PROPERTY

METHOD PUBLIC MakeReferenceTo
VAR_INPUT
	ReferenceTarget : REFERENCE TO TcVnSize2_DINT;
END_VAR
activeData REF= ReferenceTarget;
SetMemberReference();
END_METHOD

METHOD PROTECTED SetMemberReference
VAR_INPUT
END_VAR
_nWidth.MakeReferenceTo(activeData.nWidth);
_nHeight.MakeReferenceTo(activeData.nHeight);
END_METHOD

PROPERTY PUBLIC Size : UDINT
GET
Size := SIZEOF(activeData);
END_GET
END_PROPERTY

METHOD TryMakeReferenceTo : BOOL
VAR_INPUT
	Target : I_Datatype;
END_VAR
VAR
	pTargetData : POINTER TO TcVnSize2_DINT;
END_VAR
IF NOT IsEquivalentTo(Target) THEN
	RETURN;
END_IF

pTargetData := Target.Address;
activeData REF= pTargetData^;
SetMemberReference();
TryMakeReferenceTo := TRUE;
END_METHOD

PROPERTY PUBLIC Value : REFERENCE TO TcVnSize2_DINT
GET
Value REF= activeData;
END_GET
END_PROPERTY

PROPERTY PUBLIC nWidth : REFERENCE TO _DINT
GET
nWidth REF= _nWidth;
END_GET
END_PROPERTY

PROPERTY PUBLIC nHeight : REFERENCE TO _DINT
GET
nHeight REF= _nHeight;
END_GET
END_PROPERTY

END_FUNCTION_BLOCK

// ---- Datatypes/Structs/_TcVnParamsFindRois.TcPOU
{attribute 'linkalways'}
{attribute 'no_explicit_call' := 'This FB is a CLASS and must be accessed using methods or properties'}
{attribute 'enable_dynamic_creation'}
FUNCTION_BLOCK _TcVnParamsFindRois EXTENDS StructuredDatatypeBase
VAR
    localData : TcVnParamsFindRois := (stRoiSize := (nWidth := 416, nHeight := 416), fMinDensity := 0.2, fDetectionScaleFactor := 0.25, fMaxOversizeFraction := 1.0);
    activeData : REFERENCE TO TcVnParamsFindRois REF= localData;
    _stRoiSize : _TcVnSize2_DINT;
    _fMinDensity : _LREAL(localData.fMinDensity);
    _fDetectionScaleFactor : _LREAL(localData.fDetectionScaleFactor);
    _fMaxOversizeFraction : _LREAL(localData.fMaxOversizeFraction);
END_VAR

PROPERTY PUBLIC Address : PVOID
GET
Address := ADR(activeData);
END_GET
END_PROPERTY

METHOD PUBLIC ClearReference
VAR_INPUT
END_VAR
activeData REF= localData;
SetMemberReference();
END_METHOD

METHOD PUBLIC Clone : I_Datatype
VAR
    pClone : POINTER TO _TcVnParamsFindRois;
END_VAR
pClone := __NEW(_TcVnParamsFindRois);
IF pClone = 0 THEN
    RETURN;
END_IF
pClone^.TryCopyFrom(THIS^);
Clone := pClone^;
END_METHOD

METHOD FB_init : BOOL
VAR_INPUT
	bInitRetains : BOOL; // if TRUE, the retain variables are initialized (warm start / cold start)
	bInCopyCode : BOOL;  // if TRUE, the instance afterwards gets moved into the copy code (online change)
END_VAR
SetMemberReference();
AddMember('stRoiSize', _stRoiSize);
AddMember('fMinDensity', _fMinDensity);
AddMember('fDetectionScaleFactor', _fDetectionScaleFactor);
AddMember('fMaxOversizeFraction', _fMaxOversizeFraction);
END_METHOD

PROPERTY PUBLIC Identifier : T_MAXSTRING
GET
Identifier := 'TcVnParamsFindRois';
END_GET
END_PROPERTY

METHOD PUBLIC MakeReferenceTo
VAR_INPUT
	ReferenceTarget : REFERENCE TO TcVnParamsFindRois;
END_VAR
activeData REF= ReferenceTarget;
SetMemberReference();
END_METHOD

METHOD PROTECTED SetMemberReference
VAR_INPUT
END_VAR
_stRoiSize.MakeReferenceTo(activeData.stRoiSize);
_fMinDensity.MakeReferenceTo(activeData.fMinDensity);
_fDetectionScaleFactor.MakeReferenceTo(activeData.fDetectionScaleFactor);
_fMaxOversizeFraction.MakeReferenceTo(activeData.fMaxOversizeFraction);
END_METHOD

PROPERTY PUBLIC Size : UDINT
GET
Size := SIZEOF(activeData);
END_GET
END_PROPERTY

METHOD TryMakeReferenceTo : BOOL
VAR_INPUT
	Target : I_Datatype;
END_VAR
VAR
	pTargetData : POINTER TO TcVnParamsFindRois;
END_VAR
IF NOT IsEquivalentTo(Target) THEN
	RETURN;
END_IF

pTargetData := Target.Address;
activeData REF= pTargetData^;
SetMemberReference();
TryMakeReferenceTo := TRUE;
END_METHOD

PROPERTY PUBLIC Value : REFERENCE TO TcVnParamsFindRois
GET
Value REF= activeData;
END_GET
END_PROPERTY

PROPERTY PUBLIC stRoiSize : REFERENCE TO _TcVnSize2_DINT
GET
stRoiSize REF= _stRoiSize;
END_GET
END_PROPERTY

PROPERTY PUBLIC fMinDensity : REFERENCE TO _LREAL
GET
fMinDensity REF= _fMinDensity;
END_GET
END_PROPERTY

PROPERTY PUBLIC fDetectionScaleFactor : REFERENCE TO _LREAL
GET
fDetectionScaleFactor REF= _fDetectionScaleFactor;
END_GET
END_PROPERTY

PROPERTY PUBLIC fMaxOversizeFraction : REFERENCE TO _LREAL
GET
fMaxOversizeFraction REF= _fMaxOversizeFraction;
END_GET
END_PROPERTY

END_FUNCTION_BLOCK

// ---- Datatypes/Structs/_TcVnParamsWalshBarcodeDetection.TcPOU
{attribute 'linkalways'}
{attribute 'no_explicit_call' := 'This FB is a CLASS and must be accessed using methods or properties'}
{attribute 'enable_dynamic_creation'}
FUNCTION_BLOCK _TcVnParamsWalshBarcodeDetection EXTENDS StructuredDatatypeBase
VAR
    localData : TcVnParamsWalshBarcodeDetection := (nMaxBarDistance := 8, fMinAspectRatio := 1.0, fMaxAspectRatio := 5.0, nIntensityDifference := 100, nMinArea := -1, nChannelIndex := -1, nWalshFilterNum := 5, fOutlierReductionFactor := 1.0, fBarConnectionFactor := 1.0, fRegionFilterFactor := 1.0, fPostProcessingResizeFactor := 0.5, eInterpolationType := TCVN_IT_BILINEAR);
    activeData : REFERENCE TO TcVnParamsWalshBarcodeDetection REF= localData;
    _nMaxBarDistance : _UDINT(localData.nMaxBarDistance);
    _fMinAspectRatio : _REAL(localData.fMinAspectRatio);
    _fMaxAspectRatio : _REAL(localData.fMaxAspectRatio);
    _nIntensityDifference : _UDINT(localData.nIntensityDifference);
    _nMinArea : _DINT(localData.nMinArea);
    _nChannelIndex : _DINT(localData.nChannelIndex);
    _nWalshFilterNum : _UDINT(localData.nWalshFilterNum);
    _fOutlierReductionFactor : _REAL(localData.fOutlierReductionFactor);
    _fBarConnectionFactor : _REAL(localData.fBarConnectionFactor);
    _fRegionFilterFactor : _REAL(localData.fRegionFilterFactor);
    _fPostProcessingResizeFactor : _REAL(localData.fPostProcessingResizeFactor);
    _eInterpolationType : _ETcVnInterpolationType(localData.eInterpolationType);
END_VAR

PROPERTY PUBLIC Address : PVOID
GET
Address := ADR(activeData);
END_GET
END_PROPERTY

METHOD PUBLIC ClearReference
VAR_INPUT
END_VAR
activeData REF= localData;
SetMemberReference();
END_METHOD

METHOD PUBLIC Clone : I_Datatype
VAR
    pClone : POINTER TO _TcVnParamsWalshBarcodeDetection;
END_VAR
pClone := __NEW(_TcVnParamsWalshBarcodeDetection);
IF pClone = 0 THEN
    RETURN;
END_IF
pClone^.TryCopyFrom(THIS^);
Clone := pClone^;
END_METHOD

METHOD FB_init : BOOL
VAR_INPUT
	bInitRetains : BOOL; // if TRUE, the retain variables are initialized (warm start / cold start)
	bInCopyCode : BOOL;  // if TRUE, the instance afterwards gets moved into the copy code (online change)
END_VAR
SetMemberReference();
AddMember('nMaxBarDistance', _nMaxBarDistance);
AddMember('fMinAspectRatio', _fMinAspectRatio);
AddMember('fMaxAspectRatio', _fMaxAspectRatio);
AddMember('nIntensityDifference', _nIntensityDifference);
AddMember('nMinArea', _nMinArea);
AddMember('nChannelIndex', _nChannelIndex);
AddMember('nWalshFilterNum', _nWalshFilterNum);
AddMember('fOutlierReductionFactor', _fOutlierReductionFactor);
AddMember('fBarConnectionFactor', _fBarConnectionFactor);
AddMember('fRegionFilterFactor', _fRegionFilterFactor);
AddMember('fPostProcessingResizeFactor', _fPostProcessingResizeFactor);
AddMember('eInterpolationType', _eInterpolationType);
END_METHOD

PROPERTY PUBLIC Identifier : T_MAXSTRING
GET
Identifier := 'TcVnParamsWalshBarcodeDetection';
END_GET
END_PROPERTY

METHOD PUBLIC MakeReferenceTo
VAR_INPUT
	ReferenceTarget : REFERENCE TO TcVnParamsWalshBarcodeDetection;
END_VAR
activeData REF= ReferenceTarget;
SetMemberReference();
END_METHOD

METHOD PROTECTED SetMemberReference
VAR_INPUT
END_VAR
_nMaxBarDistance.MakeReferenceTo(activeData.nMaxBarDistance);
_fMinAspectRatio.MakeReferenceTo(activeData.fMinAspectRatio);
_fMaxAspectRatio.MakeReferenceTo(activeData.fMaxAspectRatio);
_nIntensityDifference.MakeReferenceTo(activeData.nIntensityDifference);
_nMinArea.MakeReferenceTo(activeData.nMinArea);
_nChannelIndex.MakeReferenceTo(activeData.nChannelIndex);
_nWalshFilterNum.MakeReferenceTo(activeData.nWalshFilterNum);
_fOutlierReductionFactor.MakeReferenceTo(activeData.fOutlierReductionFactor);
_fBarConnectionFactor.MakeReferenceTo(activeData.fBarConnectionFactor);
_fRegionFilterFactor.MakeReferenceTo(activeData.fRegionFilterFactor);
_fPostProcessingResizeFactor.MakeReferenceTo(activeData.fPostProcessingResizeFactor);
_eInterpolationType.MakeReferenceTo(activeData.eInterpolationType);
END_METHOD

PROPERTY PUBLIC Size : UDINT
GET
Size := SIZEOF(activeData);
END_GET
END_PROPERTY

METHOD TryMakeReferenceTo : BOOL
VAR_INPUT
	Target : I_Datatype;
END_VAR
VAR
	pTargetData : POINTER TO TcVnParamsWalshBarcodeDetection;
END_VAR
IF NOT IsEquivalentTo(Target) THEN
	RETURN;
END_IF

pTargetData := Target.Address;
activeData REF= pTargetData^;
SetMemberReference();
TryMakeReferenceTo := TRUE;
END_METHOD

PROPERTY PUBLIC Value : REFERENCE TO TcVnParamsWalshBarcodeDetection
GET
Value REF= activeData;
END_GET
END_PROPERTY

PROPERTY PUBLIC nMaxBarDistance : REFERENCE TO _UDINT
GET
nMaxBarDistance REF= _nMaxBarDistance;
END_GET
END_PROPERTY

PROPERTY PUBLIC fMinAspectRatio : REFERENCE TO _REAL
GET
fMinAspectRatio REF= _fMinAspectRatio;
END_GET
END_PROPERTY

PROPERTY PUBLIC fMaxAspectRatio : REFERENCE TO _REAL
GET
fMaxAspectRatio REF= _fMaxAspectRatio;
END_GET
END_PROPERTY

PROPERTY PUBLIC nIntensityDifference : REFERENCE TO _UDINT
GET
nIntensityDifference REF= _nIntensityDifference;
END_GET
END_PROPERTY

PROPERTY PUBLIC nMinArea : REFERENCE TO _DINT
GET
nMinArea REF= _nMinArea;
END_GET
END_PROPERTY

PROPERTY PUBLIC nChannelIndex : REFERENCE TO _DINT
GET
nChannelIndex REF= _nChannelIndex;
END_GET
END_PROPERTY

PROPERTY PUBLIC nWalshFilterNum : REFERENCE TO _UDINT
GET
nWalshFilterNum REF= _nWalshFilterNum;
END_GET
END_PROPERTY

PROPERTY PUBLIC fOutlierReductionFactor : REFERENCE TO _REAL
GET
fOutlierReductionFactor REF= _fOutlierReductionFactor;
END_GET
END_PROPERTY

PROPERTY PUBLIC fBarConnectionFactor : REFERENCE TO _REAL
GET
fBarConnectionFactor REF= _fBarConnectionFactor;
END_GET
END_PROPERTY

PROPERTY PUBLIC fRegionFilterFactor : REFERENCE TO _REAL
GET
fRegionFilterFactor REF= _fRegionFilterFactor;
END_GET
END_PROPERTY

PROPERTY PUBLIC fPostProcessingResizeFactor : REFERENCE TO _REAL
GET
fPostProcessingResizeFactor REF= _fPostProcessingResizeFactor;
END_GET
END_PROPERTY

PROPERTY PUBLIC eInterpolationType : REFERENCE TO _ETcVnInterpolationType
GET
eInterpolationType REF= _eInterpolationType;
END_GET
END_PROPERTY

END_FUNCTION_BLOCK

// ---- Extensions/PreExecutionCheck/PreExecutionCheckExtension.TcPOU
FUNCTION_BLOCK PreExecutionCheckExtension EXTENDS Extension
VAR
	parentAsPreCheckedNode : I_PreCheckedNode;
	preExecutionCheckFailedAlarm : PreExecutionCheckFailedAlarm(THIS^);
	enable : _BOOL(TRUE);
END_VAR

METHOD PUBLIC Check : BOOL
VAR_INPUT
END_VAR
VAR
	preExecutionChecks : PreExecutionChecks;
END_VAR
IF NOT enable.Value THEN
	IF preExecutionCheckFailedAlarm.Active THEN
		preExecutionCheckFailedAlarm.Clear();
	END_IF
	Check := TRUE;
	RETURN;
END_IF

parentAsPreCheckedNode.PreExecutionCheck(preExecutionChecks);
IF preExecutionChecks.Failed THEN
	preExecutionCheckFailedAlarm.Raise(preExecutionChecks.Reason);
	RETURN;
END_IF

preExecutionCheckFailedAlarm.Clear();
Check := TRUE;
END_METHOD

METHOD FB_init : BOOL
VAR_INPUT
	bInitRetains : BOOL; // if TRUE, the retain variables are initialized (warm start / cold start)
	bInCopyCode : BOOL;  // if TRUE, the instance afterwards gets moved into the copy code (online change)
	Name : T_MAXSTRING;
	Parent : I_HostExtensions;
END_VAR
AddParameter('enable', enable);

IF NOT __QUERYINTERFACE(Parent, parentAsPreCheckedNode) THEN
	RETURN;
END_IF
END_METHOD

END_FUNCTION_BLOCK

// ---- Extensions/WatchdogCheck/WatchdogCheckExtension.TcPOU
FUNCTION_BLOCK WatchdogCheckExtension EXTENDS Extension
VAR
	watchdogAlarm : FunctionFailedAlarm(THIS^);
	watchdogTimeInUs : _DINT(500000); // default
	hResult : HRESULT;
END_VAR

METHOD FB_init : BOOL
VAR_INPUT
	bInitRetains : BOOL; // if TRUE, the retain variables are initialized (warm start / cold start)
	bInCopyCode : BOOL;  // if TRUE, the instance afterwards gets moved into the copy code (online change)
	Name : T_MAXSTRING;
	Parent : I_HostExtensions;
END_VAR
AddParameter('watchdogTimeInUs', watchdogTimeInUs);
END_METHOD

METHOD PUBLIC Start
VAR_INPUT
END_VAR
watchdogAlarm.Clear();

IF watchdogTimeInUs.Value = 0 THEN
	RETURN;
END_IF

hResult := F_VN_StartRelWatchdog(watchdogTimeInUs.Value, S_OK);
END_METHOD

METHOD PUBLIC Stop
VAR_INPUT
END_VAR
hresult := F_VN_StopWatchdog(
	hrStartWatchdog := hresult);

IF FAILED(hresult) THEN
	watchdogAlarm.Raise('Watchdog', hresult);
END_IF
END_METHOD

END_FUNCTION_BLOCK

// ---- Functions/Checks/ContainersHaveMatchingNumberOfElements.TcPOU
FUNCTION ContainersHaveMatchingNumberOfElements : BOOL
VAR_INPUT
	Container1 : ITcVnContainer;
	Container2 : ITcVnContainer;
END_VAR
VAR
    elementNum1 : ULINT;
    elementNum2 : ULINT;
END_VAR

IF NOT IsValidContainer(Container1) THEN
	RETURN;
END_IF

IF NOT IsValidContainer(Container2) THEN
	RETURN;
END_IF

IF NOT SUCCEEDED(Container1.GetElementNum(elementNum1)) THEN
    RETURN;
END_IF

IF NOT SUCCEEDED(Container2.GetElementNum(elementNum2)) THEN
    RETURN;
END_IF

ContainersHaveMatchingNumberOfElements := (elementNum1 = elementNum2);

END_FUNCTION

// ---- Functions/Checks/IsValidContainer.TcPOU
FUNCTION IsValidContainer : BOOL
VAR_INPUT
    Container : ITcVnContainer;
END_VAR

IsValidContainer := Container <> 0;

END_FUNCTION

// ---- Functions/Checks/ImageHasCompatibleElementType.TcPOU
FUNCTION ImageHasCompatibleElementType : BOOL
VAR_INPUT
	Image : ITcVnImage;	
END_VAR
VAR_IN_OUT
	CompatibleElementTypes : ARRAY[*] OF ETcVnElementType;
END_VAR
VAR
	i : DINT;
END_VAR

IF NOT IsValidImage(Image) THEN
	RETURN;
END_IF

FOR i := LOWER_BOUND(CompatibleElementTypes, 1) TO UPPER_BOUND(CompatibleElementTypes, 1) DO
	IF ImageHasElementType(Image, CompatibleElementTypes[i]) THEN
		ImageHasCompatibleElementType := TRUE;
		RETURN;
	END_IF
END_FOR

END_FUNCTION

// ---- Functions/Checks/IsValidImage.TcPOU
FUNCTION IsValidImage : BOOL
VAR_INPUT
    Image : ITcVnImage;
END_VAR

IsValidImage := Image <> 0;

END_FUNCTION

// ---- Functions/Checks/ImageHasElementType.TcPOU
FUNCTION ImageHasElementType : BOOL
VAR_INPUT
	Image : ITcVnImage;
	ElementType : ETcVnElementType;
END_VAR

IF NOT IsValidImage(Image) THEN
	RETURN;
END_IF

ImageHasElementType := (ElementType = GetETcVnElementTypeFromImage(Image));

END_FUNCTION

// ---- Functions/Helpers/GetETcVnElementTypeFromImage.TcPOU
FUNCTION GetETcVnElementTypeFromImage : ETcVnElementType
VAR_INPUT
	sourceImage : ITcVnImage;
END_VAR
VAR
	pixelFormat : TcVnPixelFormat;
END_VAR

IF NOT IsValidImage(sourceImage) THEN
	RETURN;
END_IF

sourceImage.GetPixelFormat(pixelFormat);

IF pixelFormat.nElementSize = 8 AND NOT pixelFormat.bSigned THEN
	GetETcVnElementTypeFromImage := ETcVnElementType.TCVN_ET_USINT;
ELSIF pixelFormat.nElementSize = 8 AND pixelFormat.bSigned THEN
	GetETcVnElementTypeFromImage := ETcVnElementType.TCVN_ET_SINT;
ELSIF pixelFormat.nElementSize = 16 AND NOT pixelFormat.bSigned THEN
	GetETcVnElementTypeFromImage := ETcVnElementType.TCVN_ET_UINT;
ELSIF pixelFormat.nElementSize = 16 AND pixelFormat.bSigned THEN
	GetETcVnElementTypeFromImage := ETcVnElementType.TCVN_ET_INT;
ELSIF pixelFormat.nElementSize = 32 AND NOT pixelFormat.bFloat THEN
	GetETcVnElementTypeFromImage := ETcVnElementType.TCVN_ET_DINT;
ELSIF pixelFormat.nElementSize = 32 AND pixelFormat.bFloat THEN
	GetETcVnElementTypeFromImage := ETcVnElementType.TCVN_ET_REAL;
ELSIF pixelFormat.nElementSize = 64 THEN
	GetETcVnElementTypeFromImage := ETcVnElementType.TCVN_ET_LREAL;
ELSE
	GetETcVnElementTypeFromImage := ETcVnElementType.TCVN_ET_SAME_AS_SOURCE;
END_IF

END_FUNCTION

// ---- Functions/Checks/ImagesHaveMatchingChannels.TcPOU
FUNCTION ImagesHaveMatchingChannels : BOOL
VAR_INPUT
	Image1 : ITcVnImage;
	Image2 : ITcVnImage;
END_VAR
VAR
	pixelFormat1: TcVnPixelFormat;
	pixelFormat2: TcVnPixelFormat;
END_VAR

IF NOT IsValidImage(Image1) THEN
	RETURN;
END_IF

IF NOT IsValidImage(Image2) THEN
	RETURN;
END_IF

Image1.GetPixelFormat(pixelFormat1);
Image2.GetPixelFormat(pixelFormat2);

ImagesHaveMatchingChannels := (pixelFormat1.nChannels = pixelFormat2.nChannels);

END_FUNCTION

// ---- Functions/Checks/ContainersHaveMatchingTypes.TcPOU
FUNCTION ContainersHaveMatchingTypes : BOOL
VAR_INPUT
	Container1 : ITcVnContainer;
	Container2 : ITcVnContainer;
END_VAR
VAR
    guid1 : GUID;
    guid2 : GUID;
END_VAR

IF NOT IsValidContainer(Container1) THEN
	RETURN;
END_IF

IF NOT IsValidContainer(Container2) THEN
	RETURN;
END_IF

IF NOT SUCCEEDED(Container1.GetTypeGuid(guid1)) THEN
    RETURN;
END_IF

IF NOT SUCCEEDED(Container2.GetTypeGuid(guid2)) THEN
    RETURN;
END_IF

ContainersHaveMatchingTypes := GuidsEqualByVal(guid1, guid2);

END_FUNCTION

// ---- Functions/Checks/ImagesHaveMatchingPixelFormats.TcPOU
FUNCTION ImagesHaveMatchingPixelFormats : BOOL
VAR_INPUT
	Image1 : ITcVnImage;
	Image2 : ITcVnImage;
END_VAR
VAR
	pixelFormat_1: TcVnPixelFormat;
	pixelFormat_2: TcVnPixelFormat;
	pointer_1 : POINTER TO BYTE;
	pointer_2 : POINTER TO BYTE;
END_VAR

IF NOT IsValidImage(Image1) THEN
	RETURN;
END_IF

IF NOT IsValidImage(Image2) THEN
	RETURN;
END_IF

Image1.GetPixelFormat(pixelFormat_1);
Image2.GetPixelFormat(pixelFormat_2);

pointer_1 := ADR(pixelFormat_1);
pointer_2 := ADR(pixelFormat_2);

ImagesHaveMatchingPixelFormats := (MEMCMP(pointer_1, pointer_2, SIZEOF(pixelFormat_1)) = 0);

END_FUNCTION

// ---- Functions/Checks/IsImage1SizeEqualToImage2Size.TcPOU
FUNCTION IsImage1SizeEqualToImage2Size : BOOL
VAR_INPUT
    Image1 : ITcVnImage;
    Image2 : ITcVnImage;
END_VAR
VAR
    image1Width : UDINT;
    image1Height : UDINT;
    image2Width : UDINT;
    image2Height : UDINT;
END_VAR

IF NOT IsValidImage(Image1) THEN
    RETURN;
END_IF

IF NOT IsValidImage(Image2) THEN
    RETURN;
END_IF

Image1.GetWidth(image1Width);
Image1.GetHeight(image1Height);

Image2.GetWidth(image2Width);
Image2.GetHeight(image2Height);

IF (image1Width <> image2Width) OR_ELSE (image1Height <> image2Height) THEN
    RETURN;
END_IF

IsImage1SizeEqualToImage2Size := TRUE;

END_FUNCTION

// ---- Functions/Checks/IsImage1WidthEqualToImage2Width.TcPOU
FUNCTION IsImage1WidthEqualToImage2Width : BOOL
VAR_INPUT
    Image1 : ITcVnImage;
    Image2 : ITcVnImage;
END_VAR
VAR
    image1Width : UDINT;
    image2Width : UDINT;
END_VAR

IF NOT IsValidImage(Image1) THEN
    RETURN;
END_IF

IF NOT IsValidImage(Image2) THEN
    RETURN;
END_IF

Image1.GetWidth(image1Width);
Image2.GetWidth(image2Width);

IF (image1Width <> image2Width) THEN
    RETURN;
END_IF

IsImage1WidthEqualToImage2Width := TRUE;

END_FUNCTION

// ---- Functions/Checks/IsMaxValueCompatibleWithPixelDepth.TcPOU
FUNCTION IsMaxValueCompatibleWithPixelDepth : BOOL
VAR_INPUT
    Value : LREAL;
    PixelDepth : UINT;
END_VAR
VAR
    minimumAllowedValue : LREAL;
    maximumAllowedValue : LREAL;
END_VAR

CASE PixelDepth OF
    8:
        minimumAllowedValue := 0.0;
        TryConvert_USINT_TO_LREAL(DatatypeLimits.USINT_MAX_VALUE, maximumAllowedValue);
    16:
        minimumAllowedValue := 0.0;
        TryConvert_UINT_TO_LREAL(DatatypeLimits.UINT_MAX_VALUE, maximumAllowedValue);
    32:
        TryConvert_REAL_TO_LREAL(DatatypeLimits.REAL_MIN_VALUE, minimumAllowedValue);
        TryConvert_REAL_TO_LREAL(DatatypeLimits.REAL_MAX_VALUE, maximumAllowedValue);
    64:
        minimumAllowedValue := DatatypeLimits.LREAL_MIN_VALUE;
        maximumAllowedValue := DatatypeLimits.LREAL_MAX_VALUE;
ELSE
    ;
END_CASE

IF (Value < minimumAllowedValue) OR (Value > maximumAllowedValue) THEN
    RETURN;
END_IF

IsMaxValueCompatibleWithPixelDepth := TRUE;

END_FUNCTION

// ---- Functions/Checks/IsTemplateImageSmallerThanSourceImage.TcPOU
FUNCTION IsTemplateImageSmallerThanSourceImage : BOOL
VAR_INPUT
    SourceImage : ITcVnImage;
    TemplateImage : ITcVnImage;
END_VAR
VAR
    sourceWidth : UDINT;
    sourceHeight : UDINT;
    templateWidth : UDINT;
    templateHeight : UDINT;
END_VAR

IF NOT IsValidImage(SourceImage) THEN
    RETURN;
END_IF

IF NOT IsValidImage(TemplateImage) THEN
    RETURN;
END_IF

SourceImage.GetWidth(sourceWidth);
SourceImage.GetHeight(sourceHeight);
TemplateImage.GetWidth(templateWidth);
TemplateImage.GetHeight(templateHeight);

IF (templateWidth >= sourceWidth) THEN
    RETURN;
END_IF

IF (templateHeight >= sourceHeight) THEN
    RETURN;
END_IF

IsTemplateImageSmallerThanSourceImage := TRUE;

END_FUNCTION

// ---- Functions/Checks/IsRoiSizeOK_Udint.TcPOU
FUNCTION IsRoiSizeOK_Udint : BOOL
VAR_INPUT
    RoiRectangle : TcVnRectangle_UDINT;
    ImageWidth : UDINT;
    ImageHeight : UDINT;
END_VAR

IF NOT (RoiRectangle.nX < ImageWidth) THEN
	RETURN;
END_IF

IF NOT (RoiRectangle.nY < ImageHeight) THEN
	RETURN;
END_IF

IF NOT (RoiRectangle.nWidth <= (ImageWidth - RoiRectangle.nX)) THEN
	RETURN;
END_IF

IF NOT (RoiRectangle.nHeight <= (ImageHeight - RoiRectangle.nY)) THEN
	RETURN;
END_IF

IsRoiSizeOK_Udint := TRUE;

END_FUNCTION

// ---- Functions/Checks/IsRoiSizeOK_Dint.TcPOU
FUNCTION IsRoiSizeOK_Dint : BOOL
VAR_INPUT
    RoiRectangle : TcVnRectangle_DINT;
    ImageWidth : UDINT;
    ImageHeight : UDINT;
END_VAR
VAR
    width : DINT;
    height : DINT;
END_VAR

IF NOT TryConvert_UDINT_TO_DINT(ImageWidth, width) THEN
    RETURN;
END_IF

IF NOT TryConvert_UDINT_TO_DINT(ImageHeight, height) THEN
    RETURN;
END_IF

IF NOT (RoiRectangle.nX < width) THEN
	RETURN;
END_IF

IF NOT (RoiRectangle.nY < height) THEN
	RETURN;
END_IF

IF NOT (RoiRectangle.nWidth <= (width - RoiRectangle.nX)) THEN
	RETURN;
END_IF

IF NOT (RoiRectangle.nHeight <= (height - RoiRectangle.nY)) THEN
	RETURN;
END_IF

IsRoiSizeOK_Dint := TRUE;

END_FUNCTION

// ---- Functions/Checks/IsValidIterator.TcPOU
FUNCTION IsValidIterator : BOOL
VAR_INPUT
    Iterator : ITcVnIteratorBase;
END_VAR

IsValidIterator := Iterator <> 0;

END_FUNCTION

// ---- Nodes/Algebraic Container Ops/Node_F_VN_AddContainers.TcPOU
{attribute 'linkalways'} 
{attribute 'no_explicit_call' := 'This FB is a CLASS and must be accessed using methods or properties'}
{attribute 'enable_dynamic_creation'}
FUNCTION_BLOCK Node_F_VN_AddContainers EXTENDS VisionNode
VAR
    ipSrcContainer1 : _ITcVnContainer;
    ipSrcContainer2 : _ITcVnContainer;
    ipDestContainer : _ITcVnContainer;
    hrPrev : _HRESULT(S_OK);
    hresult : _HRESULT(S_OK);
END_VAR

METHOD PUBLIC  Clone : I_Node
VAR
    pNode : POINTER TO Node_F_VN_AddContainers;
END_VAR
pNode := __NEW(Node_F_VN_AddContainers);
Clone := pNode^;
END_METHOD

METHOD FB_init : BOOL
VAR_INPUT
    bInitRetains : BOOL; // if TRUE, the retain variables are initialized (warm start / cold start)
    bInCopyCode : BOOL;  // if TRUE, the instance afterwards gets moved into the copy code (online change)
END_VAR
AddInput('ipSrcContainer1', ipSrcContainer1);
AddInput('ipSrcContainer2', ipSrcContainer2);
AddInput('hrPrev', hrPrev);
AddOutput('ipDestContainer', ipDestContainer);
AddOutput('hresult',hresult);
END_METHOD

METHOD PROTECTED OnExecute
hresult.Value := F_VN_AddContainers(
    ipSrcContainer1 := ipSrcContainer1.Value,
    ipSrcContainer2 := ipSrcContainer2.Value,
    ipDestContainer := ipDestContainer.Value,
    hrPrev:= hrPrev.Value);
END_METHOD

METHOD PUBLIC PreExecutionCheck
VAR_INPUT
    Check : I_PreExecutionChecks;
END_VAR
Check.IsTrue(ipSrcContainer1.IsValid, 'ipSrcContainer1 must be a valid container');
Check.IsTrue(ipSrcContainer2.IsValid, 'ipSrcContainer2 must be a valid container');
Check.IsTrue(ContainersHaveMatchingTypes(ipSrcContainer1.Value, ipSrcContainer2.Value), 'Source containers must have matching types');
Check.IsTrue(ContainersHaveMatchingNumberOfElements(ipSrcContainer1.Value, ipSrcContainer2.Value), 'Source containers must contain the same number of elements');
END_METHOD

END_FUNCTION_BLOCK

// ---- Nodes/Algebraic Container Ops/Node_F_VN_BitwiseNotContainer.TcPOU
{attribute 'linkalways'} 
{attribute 'no_explicit_call' := 'This FB is a CLASS and must be accessed using methods or properties'}
{attribute 'enable_dynamic_creation'}
FUNCTION_BLOCK Node_F_VN_BitwiseNotContainer EXTENDS VisionNode
VAR
    ipSrcContainer : _ITcVnContainer;
    ipDestContainer : _ITcVnContainer;
    hrPrev : _HRESULT(S_OK);
    hresult : _HRESULT(S_OK);
END_VAR

METHOD PUBLIC  Clone : I_Node
VAR
    pNode : POINTER TO Node_F_VN_BitwiseNotContainer;
END_VAR
pNode := __NEW(Node_F_VN_BitwiseNotContainer);
Clone := pNode^;
END_METHOD

METHOD FB_init : BOOL
VAR_INPUT
    bInitRetains : BOOL; // if TRUE, the retain variables are initialized (warm start / cold start)
    bInCopyCode : BOOL;  // if TRUE, the instance afterwards gets moved into the copy code (online change)
END_VAR
AddInput('ipSrcContainer', ipSrcContainer);
AddInput('hrPrev', hrPrev);
AddOutput('ipDestContainer', ipDestContainer);
AddOutput('hresult',hresult);
END_METHOD

METHOD PROTECTED OnExecute
hresult.Value := F_VN_BitwiseNotContainer(
    ipSrcContainer := ipSrcContainer.Value,
    ipDestContainer := ipDestContainer.Value,
    hrPrev:= hrPrev.Value);
END_METHOD

METHOD PUBLIC PreExecutionCheck
VAR_INPUT
    Check : I_PreExecutionChecks;
END_VAR
Check.IsTrue(ipSrcContainer.IsValid, 'ipSrcContainer must be a valid container');

IF Check.Failed THEN
    RETURN;
END_IF

//TODO Need to check that container has integer values only.
// SINT, USINT, INT, UINT, DINT, UDINT, ULINT only?
END_METHOD

END_FUNCTION_BLOCK

// ---- Nodes/Algebraic Container Ops/Node_F_VN_BitwiseOrContainers.TcPOU
{attribute 'linkalways'} 
{attribute 'no_explicit_call' := 'This FB is a CLASS and must be accessed using methods or properties'}
{attribute 'enable_dynamic_creation'}
FUNCTION_BLOCK Node_F_VN_BitwiseOrContainers EXTENDS VisionNode
VAR
    ipSrcContainer1 : _ITcVnContainer;
    ipSrcContainer2 : _ITcVnContainer;
    ipDestContainer : _ITcVnContainer;
    hrPrev : _HRESULT(S_OK);
    hresult : _HRESULT(S_OK);
END_VAR

METHOD PUBLIC  Clone : I_Node
VAR
    pNode : POINTER TO Node_F_VN_BitwiseOrContainers;
END_VAR
pNode := __NEW(Node_F_VN_BitwiseOrContainers);
Clone := pNode^;
END_METHOD

METHOD FB_init : BOOL
VAR_INPUT
    bInitRetains : BOOL; // if TRUE, the retain variables are initialized (warm start / cold start)
    bInCopyCode : BOOL;  // if TRUE, the instance afterwards gets moved into the copy code (online change)
END_VAR
AddInput('ipSrcContainer1', ipSrcContainer1);
AddInput('ipSrcContainer2', ipSrcContainer2);
AddInput('hrPrev', hrPrev);
AddOutput('ipDestContainer', ipDestContainer);
AddOutput('hresult',hresult);
END_METHOD

METHOD PROTECTED OnExecute
hresult.Value := F_VN_BitwiseOrContainers(
    ipSrcContainer1 := ipSrcContainer1.Value,
    ipSrcContainer2 := ipSrcContainer2.Value,
    ipDestContainer := ipDestContainer.Value,
    hrPrev:= hrPrev.Value);
END_METHOD

METHOD PUBLIC PreExecutionCheck
VAR_INPUT
    Check : I_PreExecutionChecks;
END_VAR
Check.IsTrue(ipSrcContainer1.IsValid, 'ipSrcContainer1 must be a valid container');
Check.IsTrue(ipSrcContainer2.IsValid, 'ipSrcContainer2 must be a valid container');
Check.IsTrue(ContainersHaveMatchingTypes(ipSrcContainer1.Value, ipSrcContainer2.Value), 'Source containers must have matching types');
Check.IsTrue(ContainersHaveMatchingNumberOfElements(ipSrcContainer1.Value, ipSrcContainer2.Value), 'Source containers must contain the same number of elements');


//TODO Need to check that container has integer values only.
// SINT, USINT, INT, UINT, DINT, UDINT, ULINT only?
END_METHOD

END_FUNCTION_BLOCK

// ---- Nodes/Algebraic Container Ops/Node_F_VN_BitwiseXorContainers.TcPOU
{attribute 'linkalways'} 
{attribute 'no_explicit_call' := 'This FB is a CLASS and must be accessed using methods or properties'}
{attribute 'enable_dynamic_creation'}
FUNCTION_BLOCK Node_F_VN_BitwiseXorContainers EXTENDS VisionNode
VAR
    ipSrcContainer1 : _ITcVnContainer;
    ipSrcContainer2 : _ITcVnContainer;
    ipDestContainer : _ITcVnContainer;
    hrPrev : _HRESULT(S_OK);
    hresult : _HRESULT(S_OK);
END_VAR

METHOD PUBLIC  Clone : I_Node
VAR
    pNode : POINTER TO Node_F_VN_BitwiseXorContainers;
END_VAR
pNode := __NEW(Node_F_VN_BitwiseXorContainers);
Clone := pNode^;
END_METHOD

METHOD FB_init : BOOL
VAR_INPUT
    bInitRetains : BOOL; // if TRUE, the retain variables are initialized (warm start / cold start)
    bInCopyCode : BOOL;  // if TRUE, the instance afterwards gets moved into the copy code (online change)
END_VAR
AddInput('ipSrcContainer1', ipSrcContainer1);
AddInput('ipSrcContainer2', ipSrcContainer2);
AddInput('hrPrev', hrPrev);
AddOutput('ipDestContainer', ipDestContainer);
AddOutput('hresult',hresult);
END_METHOD

METHOD PROTECTED OnExecute
hresult.Value := F_VN_BitwiseXorContainers(
    ipSrcContainer1 := ipSrcContainer1.Value,
    ipSrcContainer2 := ipSrcContainer2.Value,
    ipDestContainer := ipDestContainer.Value,
    hrPrev:= hrPrev.Value);
END_METHOD

METHOD PUBLIC PreExecutionCheck
VAR_INPUT
    Check : I_PreExecutionChecks;
END_VAR
Check.IsTrue(ipSrcContainer1.IsValid, 'ipSrcContainer1 must be a valid container');
Check.IsTrue(ipSrcContainer2.IsValid, 'ipSrcContainer2 must be a valid container');
Check.IsTrue(ContainersHaveMatchingTypes(ipSrcContainer1.Value, ipSrcContainer2.Value), 'Source containers must have matching types');
Check.IsTrue(ContainersHaveMatchingNumberOfElements(ipSrcContainer1.Value, ipSrcContainer2.Value), 'Source containers must contain the same number of elements');

//TODO Need to check that container has integer values only.
// SINT, USINT, INT, UINT, DINT, UDINT, ULINT only?
END_METHOD

END_FUNCTION_BLOCK

// ---- Nodes/Algebraic Container Ops/Node_F_VN_DivideContainersExp.TcPOU
{attribute 'linkalways'} 
{attribute 'no_explicit_call' := 'This FB is a CLASS and must be accessed using methods or properties'}
{attribute 'enable_dynamic_creation'}
FUNCTION_BLOCK Node_F_VN_DivideContainersExp EXTENDS VisionNode
VAR
    ipSrcContainer1 : _ITcVnContainer;
    ipSrcContainer2 : _ITcVnContainer;
    ipDestContainer : _ITcVnContainer;
    nIntDivideByZeroResult : _LINT(0);
    hrPrev : _HRESULT(S_OK);
    hresult : _HRESULT(S_OK);
END_VAR

METHOD PUBLIC  Clone : I_Node
VAR
    pNode : POINTER TO Node_F_VN_DivideContainersExp;
END_VAR
pNode := __NEW(Node_F_VN_DivideContainersExp);
Clone := pNode^;
END_METHOD

METHOD FB_init : BOOL
VAR_INPUT
    bInitRetains : BOOL; // if TRUE, the retain variables are initialized (warm start / cold start)
    bInCopyCode : BOOL;  // if TRUE, the instance afterwards gets moved into the copy code (online change)
END_VAR
AddInput('ipSrcContainer1', ipSrcContainer1);
AddInput('ipSrcContainer2', ipSrcContainer2);
AddParameter('nIntDivideByZeroResult', nIntDivideByZeroResult);
AddInput('hrPrev', hrPrev);
AddOutput('ipDestContainer', ipDestContainer);
AddOutput('hresult',hresult);
END_METHOD

METHOD PROTECTED OnExecute
hresult.Value := F_VN_DivideContainersExp(
    ipSrcContainer1 := ipSrcContainer1.Value,
    ipSrcContainer2 := ipSrcContainer2.Value,
    nIntDivideByZeroResult := nIntDivideByZeroResult.Value,
    ipDestContainer := ipDestContainer.Value,
    hrPrev:= hrPrev.Value);
END_METHOD

METHOD PUBLIC PreExecutionCheck
VAR_INPUT
    Check : I_PreExecutionChecks;
END_VAR
Check.IsTrue(ipSrcContainer1.IsValid, 'ipSrcContainer1 must be a valid container');
Check.IsTrue(ipSrcContainer2.IsValid, 'ipSrcContainer2 must be a valid container');
Check.IsTrue(ContainersHaveMatchingTypes(ipSrcContainer1.Value, ipSrcContainer2.Value), 'Source containers must have matching types');
Check.IsTrue(ContainersHaveMatchingNumberOfElements(ipSrcContainer1.Value, ipSrcContainer2.Value), 'Source containers must contain the same number of elements');
END_METHOD

END_FUNCTION_BLOCK

// ---- Nodes/Algebraic Container Ops/Node_F_VN_BitwiseAndContainers.TcPOU
{attribute 'linkalways'} 
{attribute 'no_explicit_call' := 'This FB is a CLASS and must be accessed using methods or properties'}
{attribute 'enable_dynamic_creation'}
FUNCTION_BLOCK Node_F_VN_BitwiseAndContainers EXTENDS VisionNode
VAR
    ipSrcContainer1 : _ITcVnContainer;
    ipSrcContainer2 : _ITcVnContainer;
    ipDestContainer : _ITcVnContainer;
    hrPrev : _HRESULT(S_OK);
    hresult : _HRESULT(S_OK);
END_VAR

METHOD PUBLIC  Clone : I_Node
VAR
    pNode : POINTER TO Node_F_VN_BitwiseAndContainers;
END_VAR
pNode := __NEW(Node_F_VN_BitwiseAndContainers);
Clone := pNode^;
END_METHOD

METHOD FB_init : BOOL
VAR_INPUT
    bInitRetains : BOOL; // if TRUE, the retain variables are initialized (warm start / cold start)
    bInCopyCode : BOOL;  // if TRUE, the instance afterwards gets moved into the copy code (online change)
END_VAR
AddInput('ipSrcContainer1', ipSrcContainer1);
AddInput('ipSrcContainer2', ipSrcContainer2);
AddInput('hrPrev', hrPrev);
AddOutput('ipDestContainer', ipDestContainer);
AddOutput('hresult',hresult);
END_METHOD

METHOD PROTECTED OnExecute
hresult.Value := F_VN_BitwiseAndContainers(
    ipSrcContainer1 := ipSrcContainer1.Value,
    ipSrcContainer2 := ipSrcContainer2.Value,
    ipDestContainer := ipDestContainer.Value,
    hrPrev:= hrPrev.Value);
END_METHOD

METHOD PUBLIC PreExecutionCheck
VAR_INPUT
    Check : I_PreExecutionChecks;
END_VAR
Check.IsTrue(ipSrcContainer1.IsValid, 'ipSrcContainer1 must be a valid container');
Check.IsTrue(ipSrcContainer2.IsValid, 'ipSrcContainer2 must be a valid container');
Check.IsTrue(ContainersHaveMatchingTypes(ipSrcContainer1.Value, ipSrcContainer2.Value), 'Source containers must have matching types');
Check.IsTrue(ContainersHaveMatchingNumberOfElements(ipSrcContainer1.Value, ipSrcContainer2.Value), 'Source containers must contain the same number of elements');


//TODO Need to check that container has integer values only.
// SINT, USINT, INT, UINT, DINT, UDINT, ULINT only?
END_METHOD

END_FUNCTION_BLOCK

// ---- Nodes/Algebraic Container Ops/Node_F_VN_MaxContainer.TcPOU
{attribute 'linkalways'} 
{attribute 'no_explicit_call' := 'This FB is a CLASS and must be accessed using methods or properties'}
{attribute 'enable_dynamic_creation'}
FUNCTION_BLOCK Node_F_VN_MaxContainer EXTENDS VisionNode
VAR
    ipSrcContainer1 : _ITcVnContainer;
    ipSrcContainer2 : _ITcVnContainer;
    ipDestContainer : _ITcVnContainer;
    hrPrev : _HRESULT(S_OK);
    hresult : _HRESULT(S_OK);
END_VAR

METHOD PUBLIC  Clone : I_Node
VAR
    pNode : POINTER TO Node_F_VN_MaxContainer;
END_VAR
pNode := __NEW(Node_F_VN_MaxContainer);
Clone := pNode^;
END_METHOD

METHOD FB_init : BOOL
VAR_INPUT
    bInitRetains : BOOL; // if TRUE, the retain variables are initialized (warm start / cold start)
    bInCopyCode : BOOL;  // if TRUE, the instance afterwards gets moved into the copy code (online change)
END_VAR
AddInput('ipSrcContainer1', ipSrcContainer1);
AddInput('ipSrcContainer2', ipSrcContainer2);
AddInput('hrPrev', hrPrev);
AddOutput('ipDestContainer', ipDestContainer);
AddOutput('hresult',hresult);
END_METHOD

METHOD PROTECTED OnExecute
hresult.Value := F_VN_MaxContainer(
    ipSrcContainer1 := ipSrcContainer1.Value,
    ipSrcContainer2 := ipSrcContainer2.Value,
    ipDestContainer := ipDestContainer.Value,
    hrPrev:= hrPrev.Value);
END_METHOD

METHOD PUBLIC PreExecutionCheck
VAR_INPUT
    Check : I_PreExecutionChecks;
END_VAR
Check.IsTrue(ipSrcContainer1.IsValid, 'ipSrcContainer1 must be a valid container');
Check.IsTrue(ipSrcContainer2.IsValid, 'ipSrcContainer2 must be a valid container');
Check.IsTrue(ContainersHaveMatchingTypes(ipSrcContainer1.Value, ipSrcContainer2.Value), 'Source containers must have matching types');
Check.IsTrue(ContainersHaveMatchingNumberOfElements(ipSrcContainer1.Value, ipSrcContainer2.Value), 'Source containers must contain the same number of elements');
END_METHOD

END_FUNCTION_BLOCK

// ---- Nodes/Algebraic Container Ops/Node_F_VN_MinContainer.TcPOU
{attribute 'linkalways'} 
{attribute 'no_explicit_call' := 'This FB is a CLASS and must be accessed using methods or properties'}
{attribute 'enable_dynamic_creation'}
FUNCTION_BLOCK Node_F_VN_MinContainer EXTENDS VisionNode
VAR
    ipSrcContainer1 : _ITcVnContainer;
    ipSrcContainer2 : _ITcVnContainer;
    ipDestContainer : _ITcVnContainer;
    hrPrev : _HRESULT(S_OK);
    hresult : _HRESULT(S_OK);
END_VAR

METHOD PUBLIC  Clone : I_Node
VAR
    pNode : POINTER TO Node_F_VN_MinContainer;
END_VAR
pNode := __NEW(Node_F_VN_MinContainer);
Clone := pNode^;
END_METHOD

METHOD FB_init : BOOL
VAR_INPUT
    bInitRetains : BOOL; // if TRUE, the retain variables are initialized (warm start / cold start)
    bInCopyCode : BOOL;  // if TRUE, the instance afterwards gets moved into the copy code (online change)
END_VAR
AddInput('ipSrcContainer1', ipSrcContainer1);
AddInput('ipSrcContainer2', ipSrcContainer2);
AddInput('hrPrev', hrPrev);
AddOutput('ipDestContainer', ipDestContainer);
AddOutput('hresult',hresult);
END_METHOD

METHOD PROTECTED OnExecute
hresult.Value := F_VN_MinContainer(
    ipSrcContainer1 := ipSrcContainer1.Value,
    ipSrcContainer2 := ipSrcContainer2.Value,
    ipDestContainer := ipDestContainer.Value,
    hrPrev:= hrPrev.Value);
END_METHOD

METHOD PUBLIC PreExecutionCheck
VAR_INPUT
    Check : I_PreExecutionChecks;
END_VAR
Check.IsTrue(ipSrcContainer1.IsValid, 'ipSrcContainer1 must be a valid container');
Check.IsTrue(ipSrcContainer2.IsValid, 'ipSrcContainer2 must be a valid container');
Check.IsTrue(ContainersHaveMatchingTypes(ipSrcContainer1.Value, ipSrcContainer2.Value), 'Source containers must have matching types');
Check.IsTrue(ContainersHaveMatchingNumberOfElements(ipSrcContainer1.Value, ipSrcContainer2.Value), 'Source containers must contain the same number of elements');
END_METHOD

END_FUNCTION_BLOCK

// ---- Nodes/Algebraic Container Ops/Node_F_VN_MultiplyContainers.TcPOU
{attribute 'linkalways'} 
{attribute 'no_explicit_call' := 'This FB is a CLASS and must be accessed using methods or properties'}
{attribute 'enable_dynamic_creation'}
FUNCTION_BLOCK Node_F_VN_MultiplyContainers EXTENDS VisionNode
VAR
    ipSrcContainer1 : _ITcVnContainer;
    ipSrcContainer2 : _ITcVnContainer;
    ipDestContainer : _ITcVnContainer;
    hrPrev : _HRESULT(S_OK);
    hresult : _HRESULT(S_OK);
END_VAR

METHOD PUBLIC  Clone : I_Node
VAR
    pNode : POINTER TO Node_F_VN_MultiplyContainers;
END_VAR
pNode := __NEW(Node_F_VN_MultiplyContainers);
Clone := pNode^;
END_METHOD

METHOD FB_init : BOOL
VAR_INPUT
    bInitRetains : BOOL; // if TRUE, the retain variables are initialized (warm start / cold start)
    bInCopyCode : BOOL;  // if TRUE, the instance afterwards gets moved into the copy code (online change)
END_VAR
AddInput('ipSrcContainer1', ipSrcContainer1);
AddInput('ipSrcContainer2', ipSrcContainer2);
AddInput('hrPrev', hrPrev);
AddOutput('ipDestContainer', ipDestContainer);
AddOutput('hresult',hresult);
END_METHOD

METHOD PROTECTED OnExecute
hresult.Value := F_VN_MultiplyContainers(
    ipSrcContainer1 := ipSrcContainer1.Value,
    ipSrcContainer2 := ipSrcContainer2.Value,
    ipDestContainer := ipDestContainer.Value,
    hrPrev:= hrPrev.Value);
END_METHOD

METHOD PUBLIC PreExecutionCheck
VAR_INPUT
    Check : I_PreExecutionChecks;
END_VAR
Check.IsTrue(ipSrcContainer1.IsValid, 'ipSrcContainer1 must be a valid container');
Check.IsTrue(ipSrcContainer2.IsValid, 'ipSrcContainer2 must be a valid container');
Check.IsTrue(ContainersHaveMatchingTypes(ipSrcContainer1.Value, ipSrcContainer2.Value), 'Source containers must have matching types');
Check.IsTrue(ContainersHaveMatchingNumberOfElements(ipSrcContainer1.Value, ipSrcContainer2.Value), 'Source containers must contain the same number of elements');
END_METHOD

END_FUNCTION_BLOCK

// ---- Nodes/Algebraic Container Ops/Node_F_VN_DivideContainers.TcPOU
{attribute 'linkalways'} 
{attribute 'no_explicit_call' := 'This FB is a CLASS and must be accessed using methods or properties'}
{attribute 'enable_dynamic_creation'}
FUNCTION_BLOCK Node_F_VN_DivideContainers EXTENDS VisionNode
VAR
    ipSrcContainer1 : _ITcVnContainer;
    ipSrcContainer2 : _ITcVnContainer;
    ipDestContainer : _ITcVnContainer;
    hrPrev : _HRESULT(S_OK);
    hresult : _HRESULT(S_OK);
END_VAR

METHOD PUBLIC  Clone : I_Node
VAR
    pNode : POINTER TO Node_F_VN_DivideContainers;
END_VAR
pNode := __NEW(Node_F_VN_DivideContainers);
Clone := pNode^;
END_METHOD

METHOD FB_init : BOOL
VAR_INPUT
    bInitRetains : BOOL; // if TRUE, the retain variables are initialized (warm start / cold start)
    bInCopyCode : BOOL;  // if TRUE, the instance afterwards gets moved into the copy code (online change)
END_VAR
AddInput('ipSrcContainer1', ipSrcContainer1);
AddInput('ipSrcContainer2', ipSrcContainer2);
AddInput('hrPrev', hrPrev);
AddOutput('ipDestContainer', ipDestContainer);
AddOutput('hresult',hresult);
END_METHOD

METHOD PROTECTED OnExecute
hresult.Value := F_VN_DivideContainers(
    ipSrcContainer1 := ipSrcContainer1.Value,
    ipSrcContainer2 := ipSrcContainer2.Value,
    ipDestContainer := ipDestContainer.Value,
    hrPrev:= hrPrev.Value);
END_METHOD

METHOD PUBLIC PreExecutionCheck
VAR_INPUT
    Check : I_PreExecutionChecks;
END_VAR
Check.IsTrue(ipSrcContainer1.IsValid, 'ipSrcContainer1 must be a valid container');
Check.IsTrue(ipSrcContainer2.IsValid, 'ipSrcContainer2 must be a valid container');
Check.IsTrue(ContainersHaveMatchingTypes(ipSrcContainer1.Value, ipSrcContainer2.Value), 'Source containers must have matching types');
Check.IsTrue(ContainersHaveMatchingNumberOfElements(ipSrcContainer1.Value, ipSrcContainer2.Value), 'Source containers must contain the same number of elements');
END_METHOD

END_FUNCTION_BLOCK

// ---- Nodes/Algebraic Container Ops/Node_F_VN_NegateContainer.TcPOU
{attribute 'linkalways'} 
{attribute 'no_explicit_call' := 'This FB is a CLASS and must be accessed using methods or properties'}
{attribute 'enable_dynamic_creation'}
FUNCTION_BLOCK Node_F_VN_NegateContainer EXTENDS VisionNode
VAR
    ipSrcContainer : _ITcVnContainer;
    ipDestContainer : _ITcVnContainer;
    hrPrev : _HRESULT(S_OK);
    hresult : _HRESULT(S_OK);
END_VAR

METHOD PUBLIC  Clone : I_Node
VAR
    pNode : POINTER TO Node_F_VN_NegateContainer;
END_VAR
pNode := __NEW(Node_F_VN_NegateContainer);
Clone := pNode^;
END_METHOD

METHOD FB_init : BOOL
VAR_INPUT
    bInitRetains : BOOL; // if TRUE, the retain variables are initialized (warm start / cold start)
    bInCopyCode : BOOL;  // if TRUE, the instance afterwards gets moved into the copy code (online change)
END_VAR
AddInput('ipSrcContainer', ipSrcContainer);
AddInput('hrPrev', hrPrev);
AddOutput('ipDestContainer', ipDestContainer);
AddOutput('hresult',hresult);
END_METHOD

METHOD PROTECTED OnExecute
hresult.Value := F_VN_NegateContainer(
    ipSrcContainer := ipSrcContainer.Value,
    ipDestContainer := ipDestContainer.Value,
    hrPrev:= hrPrev.Value);
END_METHOD

METHOD PUBLIC PreExecutionCheck
VAR_INPUT
    Check : I_PreExecutionChecks;
END_VAR
Check.IsTrue(ipSrcContainer.IsValid, 'ipSrcContainer must be a valid container');
END_METHOD

END_FUNCTION_BLOCK

// ---- Nodes/Algebraic Container Ops/Node_F_VN_SubtractContainers.TcPOU
{attribute 'linkalways'} 
{attribute 'no_explicit_call' := 'This FB is a CLASS and must be accessed using methods or properties'}
{attribute 'enable_dynamic_creation'}
FUNCTION_BLOCK Node_F_VN_SubtractContainers EXTENDS VisionNode
VAR
    ipSrcContainer1 : _ITcVnContainer;
    ipSrcContainer2 : _ITcVnContainer;
    ipDestContainer : _ITcVnContainer;
    hrPrev : _HRESULT(S_OK);
    hresult : _HRESULT(S_OK);
END_VAR

METHOD PUBLIC  Clone : I_Node
VAR
    pNode : POINTER TO Node_F_VN_SubtractContainers;
END_VAR
pNode := __NEW(Node_F_VN_SubtractContainers);
Clone := pNode^;
END_METHOD

METHOD FB_init : BOOL
VAR_INPUT
    bInitRetains : BOOL; // if TRUE, the retain variables are initialized (warm start / cold start)
    bInCopyCode : BOOL;  // if TRUE, the instance afterwards gets moved into the copy code (online change)
END_VAR
AddInput('ipSrcContainer1', ipSrcContainer1);
AddInput('ipSrcContainer2', ipSrcContainer2);
AddInput('hrPrev', hrPrev);
AddOutput('ipDestContainer', ipDestContainer);
AddOutput('hresult',hresult);
END_METHOD

METHOD PROTECTED OnExecute
hresult.Value := F_VN_SubtractContainers(
    ipSrcContainer1 := ipSrcContainer1.Value,
    ipSrcContainer2 := ipSrcContainer2.Value,
    ipDestContainer := ipDestContainer.Value,
    hrPrev:= hrPrev.Value);
END_METHOD

METHOD PUBLIC PreExecutionCheck
VAR_INPUT
    Check : I_PreExecutionChecks;
END_VAR
Check.IsTrue(ipSrcContainer1.IsValid, 'ipSrcContainer1 must be a valid container');
Check.IsTrue(ipSrcContainer2.IsValid, 'ipSrcContainer2 must be a valid container');
Check.IsTrue(ContainersHaveMatchingTypes(ipSrcContainer1.Value, ipSrcContainer2.Value), 'Source containers must have matching types');
Check.IsTrue(ContainersHaveMatchingNumberOfElements(ipSrcContainer1.Value, ipSrcContainer2.Value), 'Source containers must contain the same number of elements');
END_METHOD

END_FUNCTION_BLOCK

// ---- Nodes/Algebraic Image Ops/Node_F_VN_AddImages.TcPOU
{attribute 'linkalways'} 
{attribute 'no_explicit_call' := 'This FB is a CLASS and must be accessed using methods or properties'}
{attribute 'enable_dynamic_creation'}
FUNCTION_BLOCK Node_F_VN_AddImages EXTENDS VisionNode
VAR
    ipSrcImage1 : _ITcVnImage;
    ipSrcImage2 : _ITcVnImage;
    ipDestImage : _ITcVnImage;
    hrPrev : _HRESULT(S_OK);
	hresult : _HRESULT(S_OK);
END_VAR

METHOD PUBLIC  Clone : I_Node
VAR
	pNode : POINTER TO Node_F_VN_AddImages;
END_VAR
pNode := __NEW(Node_F_VN_AddImages);
Clone := pNode^;
END_METHOD

METHOD FB_init : BOOL
VAR_INPUT
	bInitRetains : BOOL; // if TRUE, the retain variables are initialized (warm start / cold start)
	bInCopyCode : BOOL;  // if TRUE, the instance afterwards gets moved into the copy code (online change)
END_VAR
AddInput('ipSrcImage1', ipSrcImage1);
AddInput('ipSrcImage2', ipSrcImage2);
AddInput('hrPrev', hrPrev);
AddOutput('ipDestImage', ipDestImage);
AddOutput('hresult',hresult);
END_METHOD

METHOD PROTECTED OnExecute
hresult.Value := F_VN_AddImages(
    ipSrcImage1 := ipSrcImage1.Value,
    ipSrcImage2 := ipSrcImage2.Value,
	ipDestImage := ipDestImage.Value,
	hrPrev:= hrPrev.Value);
END_METHOD

METHOD PUBLIC PreExecutionCheck
VAR_INPUT
	Check : I_PreExecutionChecks;
END_VAR
Check.IsTrue(ipSrcImage1.IsValid, 'ipSrcImage1 must contain an image');
Check.IsTrue(ipSrcImage2.IsValid, 'ipSrcImage2 must contain an image');
Check.IsTrue(IsImage1SizeEqualToImage2Size(ipSrcImage1.Value, ipSrcImage2.Value), 'ipSrcImage1 must be the same size as ipSrcImage2');
END_METHOD

END_FUNCTION_BLOCK

// ---- Nodes/Algebraic Image Ops/Node_F_VN_AddImagesWeighted.TcPOU
{attribute 'linkalways'} 
{attribute 'no_explicit_call' := 'This FB is a CLASS and must be accessed using methods or properties'}
{attribute 'enable_dynamic_creation'}
FUNCTION_BLOCK Node_F_VN_AddImagesWeighted EXTENDS VisionNode
VAR
    ipSrcImage1 : _ITcVnImage;
    ipSrcImage2 : _ITcVnImage;
    ipDestImage : _ITcVnImage;
    fWeight1 : _LREAL(0.0);
    fWeight2 : _LREAL(0.0);
    fDelta : _LREAL(0.0);
    hrPrev : _HRESULT(S_OK);
	hresult : _HRESULT(S_OK);
END_VAR

METHOD PUBLIC  Clone : I_Node
VAR
	pNode : POINTER TO Node_F_VN_AddImagesWeighted;
END_VAR
pNode := __NEW(Node_F_VN_AddImagesWeighted);
Clone := pNode^;
END_METHOD

METHOD FB_init : BOOL
VAR_INPUT
	bInitRetains : BOOL; // if TRUE, the retain variables are initialized (warm start / cold start)
	bInCopyCode : BOOL;  // if TRUE, the instance afterwards gets moved into the copy code (online change)
END_VAR
AddInput('ipSrcImage1', ipSrcImage1);
AddInput('ipSrcImage2', ipSrcImage2);
AddParameter('fWeight1', fWeight1);
AddParameter('fWeight2', fWeight2);
AddParameter('fDelta', fDelta);
AddInput('hrPrev', hrPrev);
AddOutput('ipDestImage', ipDestImage);
AddOutput('hresult',hresult);
END_METHOD

METHOD PROTECTED OnExecute
hresult.Value := F_VN_AddImagesWeighted(
    ipSrcImage1 := ipSrcImage1.Value,
    ipSrcImage2 := ipSrcImage2.Value,
	ipDestImage := ipDestImage.Value,
    fWeight1 := fWeight1.Value,
    fWeight2 := fWeight2.Value,
    fDelta := fDelta.Value,
	hrPrev:= hrPrev.Value);
END_METHOD

METHOD PUBLIC PreExecutionCheck
VAR_INPUT
	Check : I_PreExecutionChecks;
END_VAR
Check.IsTrue(ipSrcImage1.IsValid, 'ipSrcImage1 must contain an image');
Check.IsTrue(ipSrcImage2.IsValid, 'ipSrcImage2 must contain an image');
Check.IsTrue(IsImage1SizeEqualToImage2Size(ipSrcImage1.Value, ipSrcImage2.Value), 'ipSrcImage1 must be the same size as ipSrcImage2');
END_METHOD

END_FUNCTION_BLOCK

// ---- Nodes/Algebraic Image Ops/Node_F_VN_AddImagesWeightedExp.TcPOU
{attribute 'linkalways'} 
{attribute 'no_explicit_call' := 'This FB is a CLASS and must be accessed using methods or properties'}
{attribute 'enable_dynamic_creation'}
FUNCTION_BLOCK Node_F_VN_AddImagesWeightedExp EXTENDS VisionNode
VAR
    ipSrcImage1 : _ITcVnImage;
    ipSrcImage2 : _ITcVnImage;
    ipDestImage : _ITcVnImage;
    fWeight1 : _LREAL(0.0);
    fWeight2 : _LREAL(0.0);
    fDelta : _LREAL(0.0);
    eDestType : _ETcVnElementType(ETcVnElementType.TCVN_ET_SAME_AS_SOURCE);
    hrPrev : _HRESULT(S_OK);
	hresult : _HRESULT(S_OK);
END_VAR

METHOD PUBLIC  Clone : I_Node
VAR
	pNode : POINTER TO Node_F_VN_AddImagesWeightedExp;
END_VAR
pNode := __NEW(Node_F_VN_AddImagesWeightedExp);
Clone := pNode^;
END_METHOD

METHOD FB_init : BOOL
VAR_INPUT
	bInitRetains : BOOL; // if TRUE, the retain variables are initialized (warm start / cold start)
	bInCopyCode : BOOL;  // if TRUE, the instance afterwards gets moved into the copy code (online change)
END_VAR
AddInput('ipSrcImage1', ipSrcImage1);
AddInput('ipSrcImage2', ipSrcImage2);
AddParameter('fWeight1', fWeight1);
AddParameter('fWeight2', fWeight2);
AddParameter('fDelta', fDelta);
AddParameter('eDestType', eDestType);
AddInput('hrPrev', hrPrev);
AddOutput('ipDestImage', ipDestImage);
AddOutput('hresult',hresult);
END_METHOD

METHOD PROTECTED OnExecute
hresult.Value := F_VN_AddImagesWeightedExp(
    ipSrcImage1 := ipSrcImage1.Value,
    ipSrcImage2 := ipSrcImage2.Value,
	ipDestImage := ipDestImage.Value,
    fWeight1 := fWeight1.Value,
    fWeight2 := fWeight2.Value,
    fDelta := fDelta.Value,
    eDestType := eDestType.Value,
	hrPrev:= hrPrev.Value);
END_METHOD

METHOD PUBLIC PreExecutionCheck
VAR_INPUT
	Check : I_PreExecutionChecks;
END_VAR
Check.IsTrue(ipSrcImage1.IsValid, 'ipSrcImage1 must contain an image');
Check.IsTrue(ipSrcImage2.IsValid, 'ipSrcImage2 must contain an image');
Check.IsTrue(IsImage1SizeEqualToImage2Size(ipSrcImage1.Value, ipSrcImage2.Value), 'ipSrcImage1 must be the same size as ipSrcImage2');
END_METHOD

END_FUNCTION_BLOCK

// ---- Nodes/Algebraic Image Ops/Node_F_VN_AddVectorToImage.TcPOU
{attribute 'linkalways'} 
{attribute 'no_explicit_call' := 'This FB is a CLASS and must be accessed using methods or properties'}
{attribute 'enable_dynamic_creation'}
FUNCTION_BLOCK Node_F_VN_AddVectorToImage EXTENDS VisionNode
VAR
    aVector : _TcVnVector4_LREAL;
    ipSrcImage : _ITcVnImage;
    ipDestImage : _ITcVnImage;
    hrPrev : _HRESULT(S_OK);
	hresult : _HRESULT(S_OK);
END_VAR

METHOD PUBLIC  Clone : I_Node
VAR
	pNode : POINTER TO Node_F_VN_AddVectorToImage;
END_VAR
pNode := __NEW(Node_F_VN_AddVectorToImage);
Clone := pNode^;
END_METHOD

METHOD FB_init : BOOL
VAR_INPUT
	bInitRetains : BOOL; // if TRUE, the retain variables are initialized (warm start / cold start)
	bInCopyCode : BOOL;  // if TRUE, the instance afterwards gets moved into the copy code (online change)
END_VAR
AddInput('aVector', aVector);
AddInput('ipSrcImage', ipSrcImage);
AddInput('hrPrev', hrPrev);
AddOutput('ipDestImage', ipDestImage);
AddOutput('hresult',hresult);
END_METHOD

METHOD PROTECTED OnExecute
hresult.Value := F_VN_AddVectorToImage(
    aVector := aVector.Value,
    ipSrcImage := ipSrcImage.Value,
	ipDestImage := ipDestImage.Value,
	hrPrev:= hrPrev.Value);
END_METHOD

METHOD PUBLIC PreExecutionCheck
VAR_INPUT
	Check : I_PreExecutionChecks;
END_VAR
Check.IsTrue(ipSrcImage.IsValid, 'ipSrcImage must contain an image');
END_METHOD

END_FUNCTION_BLOCK

// ---- Nodes/Algebraic Image Ops/Node_F_VN_BitwiseAndImagesExp.TcPOU
{attribute 'linkalways'} 
{attribute 'no_explicit_call' := 'This FB is a CLASS and must be accessed using methods or properties'}
{attribute 'enable_dynamic_creation'}
FUNCTION_BLOCK Node_F_VN_BitwiseAndImagesExp EXTENDS VisionNode
VAR
    ipSrcImage1 : _ITcVnImage;
    ipSrcImage2 : _ITcVnImage;
    ipDestImage : _ITcVnImage;
    ipMask : _ITcVnImage;
    hrPrev : _HRESULT(S_OK);
	hresult : _HRESULT(S_OK);
END_VAR

METHOD PUBLIC  Clone : I_Node
VAR
	pNode : POINTER TO Node_F_VN_BitwiseAndImagesExp;
END_VAR
pNode := __NEW(Node_F_VN_BitwiseAndImagesExp);
Clone := pNode^;
END_METHOD

METHOD FB_init : BOOL
VAR_INPUT
	bInitRetains : BOOL; // if TRUE, the retain variables are initialized (warm start / cold start)
	bInCopyCode : BOOL;  // if TRUE, the instance afterwards gets moved into the copy code (online change)
END_VAR
AddInput('ipSrcImage1', ipSrcImage1);
AddInput('ipSrcImage2', ipSrcImage2);
AddInput('ipMask', ipMask);
AddInput('hrPrev', hrPrev);
AddOutput('ipDestImage', ipDestImage);
AddOutput('hresult',hresult);
END_METHOD

METHOD PROTECTED OnExecute
hresult.Value := F_VN_BitwiseAndImagesExp(
    ipSrcImage1 := ipSrcImage1.Value,
    ipSrcImage2 := ipSrcImage2.Value,
	ipDestImage := ipDestImage.Value,
    ipMask := ipMask.Value,
	hrPrev:= hrPrev.Value);
END_METHOD

METHOD PUBLIC PreExecutionCheck
VAR_INPUT
	Check : I_PreExecutionChecks;
END_VAR
Check.IsTrue(ipSrcImage1.IsValid, 'ipSrcImage1 must contain an image');
Check.IsTrue(ipSrcImage2.IsValid, 'ipSrcImage2 must contain an image');
Check.IsTrue(IsImage1SizeEqualToImage2Size(ipSrcImage1.Value, ipSrcImage2.Value), 'ipSrcImage1 must be the same size as ipSrcImage2');
Check.IsTrue(ipMask.IsValid, 'ipMask must contain an image');
Check.IsTrue(ipMask.HasChannelCount(1), 'ipMask must have 1 channel');
Check.IsTrue(ipMask.IsPixelDepth(8), 'ipMask must have 8 bit pixel depth');
Check.IsTrue(IsImage1SizeEqualToImage2Size(ipMask.Value, ipSrcImage1.Value), 'ipMask must be the same size as ipSrcImage1');
END_METHOD

END_FUNCTION_BLOCK

// ---- Nodes/Algebraic Image Ops/Node_F_VN_BitwiseNotImageExp.TcPOU
{attribute 'linkalways'} 
{attribute 'no_explicit_call' := 'This FB is a CLASS and must be accessed using methods or properties'}
{attribute 'enable_dynamic_creation'}
FUNCTION_BLOCK Node_F_VN_BitwiseNotImageExp EXTENDS VisionNode
VAR
    ipSrcImage : _ITcVnImage;
    ipDestImage : _ITcVnImage;
    ipMask : _ITcVnImage;
    hrPrev : _HRESULT(S_OK);
	hresult : _HRESULT(S_OK);
END_VAR

METHOD PUBLIC  Clone : I_Node
VAR
	pNode : POINTER TO Node_F_VN_BitwiseNotImageExp;
END_VAR
pNode := __NEW(Node_F_VN_BitwiseNotImageExp);
Clone := pNode^;
END_METHOD

METHOD FB_init : BOOL
VAR_INPUT
	bInitRetains : BOOL; // if TRUE, the retain variables are initialized (warm start / cold start)
	bInCopyCode : BOOL;  // if TRUE, the instance afterwards gets moved into the copy code (online change)
END_VAR
AddInput('ipSrcImage', ipSrcImage);
AddInput('ipMask', ipMask);
AddInput('hrPrev', hrPrev);
AddOutput('ipDestImage', ipDestImage);
AddOutput('hresult',hresult);
END_METHOD

METHOD PROTECTED OnExecute
hresult.Value := F_VN_BitwiseNotImageExp(
    ipSrcImage := ipSrcImage.Value,
	ipDestImage := ipDestImage.Value,
    ipMask := ipMask.Value,
	hrPrev:= hrPrev.Value);
END_METHOD

METHOD PUBLIC PreExecutionCheck
VAR_INPUT
	Check : I_PreExecutionChecks;
END_VAR
Check.IsTrue(ipSrcImage.IsValid, 'ipSrcImage must contain an image');
Check.IsTrue(ipMask.IsValid, 'ipMask must contain an image');
Check.IsTrue(ipMask.HasChannelCount(1), 'ipMask must have 1 channel');
Check.IsTrue(ipMask.IsPixelDepth(8), 'ipMask must have 8 bit pixel depth');
Check.IsTrue(IsImage1SizeEqualToImage2Size(ipMask.Value, ipSrcImage.Value), 'ipMask must be the same size as ipSrcImage');
END_METHOD

END_FUNCTION_BLOCK

// ---- Nodes/Algebraic Image Ops/Node_F_VN_MaxImageExp.TcPOU
{attribute 'linkalways'} 
{attribute 'no_explicit_call' := 'This FB is a CLASS and must be accessed using methods or properties'}
{attribute 'enable_dynamic_creation'}
FUNCTION_BLOCK Node_F_VN_MaxImageExp EXTENDS VisionNode
VAR
    ipSrcImage1 : _ITcVnImage;
    ipSrcImage2 : _ITcVnImage;
    ipDestImage : _ITcVnImage;
    ipMask : _ITcVnImage;
    hrPrev : _HRESULT(S_OK);
	hresult : _HRESULT(S_OK);
END_VAR

METHOD PUBLIC  Clone : I_Node
VAR
	pNode : POINTER TO Node_F_VN_MaxImageExp;
END_VAR
pNode := __NEW(Node_F_VN_MaxImageExp);
Clone := pNode^;
END_METHOD

METHOD FB_init : BOOL
VAR_INPUT
	bInitRetains : BOOL; // if TRUE, the retain variables are initialized (warm start / cold start)
	bInCopyCode : BOOL;  // if TRUE, the instance afterwards gets moved into the copy code (online change)
END_VAR
AddInput('ipSrcImage1', ipSrcImage1);
AddInput('ipSrcImage2', ipSrcImage2);
AddInput('ipMask', ipMask);
AddInput('hrPrev', hrPrev);
AddOutput('ipDestImage', ipDestImage);
AddOutput('hresult',hresult);
END_METHOD

METHOD PROTECTED OnExecute
hresult.Value := F_VN_MaxImageExp(
    ipSrcImage1 := ipSrcImage1.Value,
    ipSrcImage2 := ipSrcImage2.Value,
	ipDestImage := ipDestImage.Value,
    ipMask := ipMask.Value,
	hrPrev:= hrPrev.Value);
END_METHOD

METHOD PUBLIC PreExecutionCheck
VAR_INPUT
	Check : I_PreExecutionChecks;
END_VAR
Check.IsTrue(ipSrcImage1.IsValid, 'ipSrcImage1 must contain an image');
Check.IsTrue(ipSrcImage2.IsValid, 'ipSrcImage2 must contain an image');
Check.IsTrue(IsImage1SizeEqualToImage2Size(ipSrcImage1.Value, ipSrcImage2.Value), 'ipSrcImage1 must be the same size as ipSrcImage2');
Check.IsTrue(ipMask.IsValid, 'ipMask must contain an image');
Check.IsTrue(ipMask.HasChannelCount(1), 'ipMask must have 1 channel');
Check.IsTrue(ipMask.IsPixelDepth(8), 'ipMask must have 8 bit pixel depth');
Check.IsTrue(IsImage1SizeEqualToImage2Size(ipMask.Value, ipSrcImage1.Value), 'ipMask must be the same size as ipSrcImage1');
END_METHOD

END_FUNCTION_BLOCK

